SPLINE
SPL {X  -165.650, Y  +484.445, Z    +0.000, E1   +32.277, E3 +434870.647}
SPL {X  -165.650, Y  +481.524, Z    +0.000, E1   +31.089, E3 +434888.097}
SPL {X  -165.650, Y  +478.014, Z    +0.000, E1   +30.826, E3 +434901.705}
SPL {X  -165.650, Y  +474.473, Z    +0.000, E1   +30.943, E3 +434913.029}
SPL {X  -165.650, Y  +471.826, Z    +0.000, E1   +30.770, E3 +434923.213}
SPL {X  -165.650, Y  +467.753, Z    +0.000, E1   +30.878, E3 +434936.586}
SPL {X  -165.650, Y  +463.837, Z    +0.000, E1   +30.924, E3 +434949.520}
SPL {X  -165.650, Y  +461.106, Z    +0.000, E1   +30.916, E3 +434958.907}
SPL {X  -165.650, Y  +457.156, Z    +0.000, E1   +30.860, E3 +434972.984}
SPL {X  -165.650, Y  +453.156, Z    +0.000, E1   +30.934, E3 +434985.958}
SPL {X  -165.650, Y  +450.433, Z    +0.000, E1   +30.789, E3 +434996.313}
SPL {X  -165.650, Y  +447.097, Z    +0.000, E1   +30.843, E3 +435007.362}
SPL {X  -165.650, Y  +443.673, Z    +0.000, E1   +30.907, E3 +435018.669}
SPL {X  -165.650, Y  +439.486, Z    +0.000, E1   +30.857, E3 +435033.479}
SPL {X  -165.650, Y  +435.146, Z    +0.000, E1   +30.969, E3 +435047.398}
SPL {X  -165.650, Y  +431.607, Z    +0.000, E1   +30.889, E3 +435060.113}
SPL {X  -165.650, Y  +427.340, Z    +0.000, E1   +30.870, E3 +435074.824}
SPL {X  -165.650, Y  +423.901, Z    +0.000, E1   +30.858, E3 +435086.580}
SPL {X  -165.650, Y  +421.437, Z    +0.000, E1   +30.833, E3 +435095.179}
SPL {X  -165.650, Y  +418.489, Z    +0.000, E1   +30.835, E3 +435105.295}
SPL {X  -165.650, Y  +414.127, Z    +0.000, E1   +30.869, E3 +435120.204}
SPL {X  -165.650, Y  +408.547, Z    +0.000, E1   +30.964, E3 +435138.620}
SPL {X  -165.650, Y  +405.433, Z    +0.000, E1   +30.730, E3 +435150.597}
SPL {X  -165.650, Y  +401.473, Z    +0.000, E1   +30.933, E3 +435163.045}
SPL {X  -165.650, Y  +396.018, Z    +0.000, E1   +30.861, E3 +435182.230}
SPL {X  -165.650, Y  +390.331, Z    +0.000, E1   +30.892, E3 +435201.483}
SPL {X  -165.650, Y  +384.849, Z    +0.000, E1   +30.885, E3 +435220.286}
SPL {X  -165.650, Y  +380.752, Z    +0.000, E1   +30.927, E3 +435233.787}
SPL {X  -165.648, Y  +377.739, Z    +0.000, E1   +30.835, E3 +435244.797}
SPL {X  -165.594, Y  +374.183, Z    +0.000, E1   +30.878, E3 +435256.634}
SPL {X  -165.492, Y  +371.263, Z    +0.000, E1   +30.913, E3 +435266.329}
SPL {X  -165.379, Y  +369.027, Z    +0.000, E1   +30.727, E3 +435275.267}
SPL {X  -165.167, Y  +365.866, Z    +0.000, E1   +30.741, E3 +435286.041}
SPL {X  -164.892, Y  +362.671, Z    +0.000, E1   +30.830, E3 +435296.365}
SPL {X  -164.570, Y  +359.612, Z    +0.000, E1   +30.773, E3 +435307.178}
SPL {X  -164.104, Y  +355.923, Z    +0.000, E1   +30.626, E3 +435320.895}
SPL {X  -163.573, Y  +352.353, Z    +0.000, E1   +30.451, E3 +435334.159}
SPL {X  -162.476, Y  +346.230, Z    +0.000, E1   +31.677, E3 +435346.740}
SPL {X  -152.976, Y  +314.952, Z    +0.000, E1   +38.607, E3 +435395.705}
SPL {X  -137.967, Y  +286.821, Z    +0.000, E1   +43.969, E3 +435438.926}
ENDSPLINE

SPLINE
SPL {X  -153.316, Y  +315.777, Z    +0.000, E1   +33.140, E3 +435481.554}
SPL {X  -164.446, Y  +358.564, Z    +0.000, E1   +15.149, E3 +435446.765}
SPL {X  -165.379, Y  +369.025, Z    +0.000, E1    +9.158, E3 +435452.490}
SPL {X  -165.612, Y  +374.969, Z    +0.000, E1    +5.630, E3 +435455.165}
SPL {X  -165.650, Y  +383.362, Z    +0.000, E1    +0.177, E3 +435439.783}
SPL {X  -165.650, Y  +383.923, Z    +0.000, E1    -0.215, E3 +435452.941}
SPL {X  -165.650, Y  +388.083, Z    +0.000, E1    -3.355, E3 +435451.804}
SPL {X  -165.650, Y  +393.983, Z    +0.000, E1    -8.501, E3 +435448.203}
SPL {X  -165.650, Y  +402.241, Z    +0.000, E1   -16.711, E3 +435442.714}
SPL {X  -165.650, Y  +416.345, Z    +0.000, E1   -29.511, E3 +435442.506}
SPL {X  -165.650, Y  +422.331, Z    +0.000, E1   -27.760, E3 +435468.005}
SPL {X  -165.650, Y  +441.276, Z    +0.000, E1   -37.343, E3 +435477.862}
SPL {X  -165.650, Y  +462.890, Z    +0.000, E1   -40.484, E3 +435511.945}
ENDSPLINE

SPLINE
SPL {X  -165.650, Y  +446.920, Z    +0.000, E1   -31.238, E3 +435524.271}
ENDSPLINE

SPLINE
SPL {X  -165.650, Y  +447.935, Z    +0.000, E1   -30.213, E3 +435534.559}
SPL {X  -165.650, Y  +451.020, Z    +0.000, E1   -30.224, E3 +435545.379}
SPL {X  -165.650, Y  +454.519, Z    +0.000, E1   -30.374, E3 +435556.562}
SPL {X  -165.650, Y  +456.542, Z    +0.000, E1   -29.986, E3 +435566.306}
SPL {X  -165.650, Y  +460.618, Z    +0.000, E1   -30.298, E3 +435578.627}
SPL {X  -165.650, Y  +463.853, Z    +0.000, E1   -30.103, E3 +435591.228}
SPL {X  -165.650, Y  +467.246, Z    +0.000, E1   -30.279, E3 +435601.958}
SPL {X  -165.650, Y  +469.780, Z    +0.000, E1   -30.237, E3 +435611.083}
SPL {X  -165.650, Y  +472.566, Z    +0.000, E1   -30.124, E3 +435621.741}
SPL {X  -165.650, Y  +476.540, Z    +0.000, E1   -30.193, E3 +435635.285}
SPL {X  -165.650, Y  +480.320, Z    +0.000, E1   -30.163, E3 +435648.763}
SPL {X  -165.650, Y  +484.477, Z    +0.000, E1   -30.274, E3 +435662.652}
SPL {X  -165.650, Y  +488.041, Z    +0.000, E1   -30.253, E3 +435675.207}
SPL {X  -165.650, Y  +491.281, Z    +0.000, E1   -30.148, E3 +435687.345}
SPL {X  -165.650, Y  +495.051, Z    +0.000, E1   -30.213, E3 +435700.154}
SPL {X  -165.650, Y  +498.418, Z    +0.000, E1   -30.282, E3 +435711.447}
SPL {X  -165.650, Y  +500.833, Z    +0.000, E1   -30.191, E3 +435720.496}
SPL {X  -165.650, Y  +504.246, Z    +0.000, E1   -30.231, E3 +435732.362}
SPL {X  -165.650, Y  +507.017, Z    +0.000, E1   -30.108, E3 +435742.771}
SPL {X  -165.650, Y  +510.660, Z    +0.000, E1   -30.223, E3 +435755.037}
SPL {X  -165.650, Y  +515.918, Z    +0.000, E1   -30.316, E3 +435772.846}
SPL {X  -165.650, Y  +520.621, Z    +0.000, E1   -30.198, E3 +435790.131}
SPL {X  -165.650, Y  +525.344, Z    +0.000, E1   -30.269, E3 +435806.187}
SPL {X  -165.650, Y  +528.152, Z    +0.000, E1   -29.991, E3 +435817.828}
SPL {X  -165.650, Y  +531.783, Z    +0.000, E1   -30.416, E3 +435827.721}
SPL {X  -165.650, Y  +534.115, Z    +0.000, E1   -30.089, E3 +435838.103}
SPL {X  -165.650, Y  +538.363, Z    +0.000, E1   -30.232, E3 +435852.273}
SPL {X  -165.650, Y  +543.650, Z    +0.000, E1   -30.281, E3 +435870.493}
SPL {X  -165.650, Y  +547.199, Z    +0.000, E1   -30.132, E3 +435883.752}
SPL {X  -165.650, Y  +550.512, Z    +0.000, E1   -30.197, E3 +435895.078}
SPL {X  -165.650, Y  +554.908, Z    +0.000, E1   -30.180, E3 +435910.739}
SPL {X  -165.650, Y  +560.243, Z    +0.000, E1   -30.214, E3 +435929.365}
SPL {X  -165.650, Y  +565.528, Z    +0.000, E1   -30.192, E3 +435948.057}
SPL {X  -165.650, Y  +570.048, Z    +0.000, E1   -30.238, E3 +435963.488}
SPL {X  -165.650, Y  +573.110, Z    +0.000, E1   -30.057, E3 +435975.473}
SPL {X  -165.650, Y  +577.587, Z    +0.000, E1   -30.270, E3 +435989.912}
SPL {X  -165.650, Y  +581.190, Z    +0.000, E1   -30.107, E3 +436003.551}
SPL {X  -165.650, Y  +585.053, Z    +0.000, E1   -30.090, E3 +436017.422}
ENDSPLINE

SPLINE
SPL {X  -165.650, Y  +484.445, Z    +0.000, E1   +32.277, E3 +436034.826}
SPL {X  -165.650, Y  +481.524, Z    +0.000, E1   +31.089, E3 +436052.277}
SPL {X  -165.650, Y  +478.014, Z    +0.000, E1   +30.826, E3 +436065.884}
SPL {X  -165.650, Y  +474.473, Z    +0.000, E1   +30.943, E3 +436077.209}
SPL {X  -165.650, Y  +471.826, Z    +0.000, E1   +30.770, E3 +436087.392}
SPL {X  -165.650, Y  +467.753, Z    +0.000, E1   +30.878, E3 +436100.766}
SPL {X  -165.650, Y  +463.837, Z    +0.000, E1   +30.924, E3 +436113.699}
SPL {X  -165.650, Y  +461.106, Z    +0.000, E1   +30.916, E3 +436123.086}
SPL {X  -165.650, Y  +457.156, Z    +0.000, E1   +30.860, E3 +436137.163}
SPL {X  -165.650, Y  +453.156, Z    +0.000, E1   +30.934, E3 +436150.137}
SPL {X  -165.650, Y  +450.433, Z    +0.000, E1   +30.789, E3 +436160.492}
SPL {X  -165.650, Y  +447.097, Z    +0.000, E1   +30.843, E3 +436171.541}
SPL {X  -165.650, Y  +443.673, Z    +0.000, E1   +30.907, E3 +436182.848}
SPL {X  -165.650, Y  +439.486, Z    +0.000, E1   +30.857, E3 +436197.658}
SPL {X  -165.650, Y  +434.043, Z    +0.000, E1   +30.950, E3 +436215.674}
SPL {X  -165.650, Y  +430.419, Z    +0.000, E1   +30.895, E3 +436228.177}
SPL {X  -165.650, Y  +427.340, Z    +0.000, E1   +30.870, E3 +436239.003}
SPL {X  -165.650, Y  +422.641, Z    +0.000, E1   +30.884, E3 +436255.092}
SPL {X  -165.650, Y  +417.366, Z    +0.000, E1   +30.879, E3 +436273.198}
SPL {X  -165.650, Y  +412.139, Z    +0.000, E1   +30.870, E3 +436291.148}
SPL {X  -165.650, Y  +406.834, Z    +0.000, E1   +30.919, E3 +436308.976}
SPL {X  -165.650, Y  +402.516, Z    +0.000, E1   +30.874, E3 +436323.899}
SPL {X  -165.650, Y  +398.147, Z    +0.000, E1   +30.902, E3 +436338.777}
SPL {X  -165.650, Y  +394.694, Z    +0.000, E1   +30.805, E3 +436351.085}
SPL {X  -165.650, Y  +391.522, Z    +0.000, E1   +30.837, E3 +436361.766}
SPL {X  -165.650, Y  +387.533, Z    +0.000, E1   +30.858, E3 +436375.392}
SPL {X  -165.650, Y  +383.627, Z    +0.000, E1   +30.885, E3 +436388.453}
SPL {X  -165.650, Y  +380.752, Z    +0.000, E1   +30.927, E3 +436397.967}
SPL {X  -165.648, Y  +377.739, Z    +0.000, E1   +30.835, E3 +436408.976}
SPL {X  -165.594, Y  +374.183, Z    +0.000, E1   +30.878, E3 +436420.813}
SPL {X  -165.492, Y  +371.263, Z    +0.000, E1   +30.913, E3 +436430.508}
SPL {X  -165.379, Y  +369.027, Z    +0.000, E1   +30.727, E3 +436439.446}
SPL {X  -165.167, Y  +365.866, Z    +0.000, E1   +30.741, E3 +436450.220}
SPL {X  -164.892, Y  +362.671, Z    +0.000, E1   +30.830, E3 +436460.545}
SPL {X  -164.570, Y  +359.612, Z    +0.000, E1   +30.773, E3 +436471.357}
SPL {X  -164.104, Y  +355.923, Z    +0.000, E1   +30.626, E3 +436485.074}
SPL {X  -163.573, Y  +352.353, Z    +0.000, E1   +30.451, E3 +436498.338}
SPL {X  -162.476, Y  +346.230, Z    +0.000, E1   +31.677, E3 +436510.919}
SPL {X  -152.976, Y  +314.952, Z    +0.000, E1   +38.607, E3 +436559.884}
SPL {X  -137.967, Y  +286.821, Z    +0.000, E1   +43.969, E3 +436603.106}
ENDSPLINE

SPLINE
SPL {X  -153.316, Y  +315.777, Z    +0.000, E1   +33.140, E3 +436645.733}
SPL {X  -164.446, Y  +358.564, Z    +0.000, E1   +15.149, E3 +436610.944}
SPL {X  -165.379, Y  +369.025, Z    +0.000, E1    +9.158, E3 +436616.669}
SPL {X  -165.612, Y  +374.969, Z    +0.000, E1    +5.630, E3 +436619.344}
SPL {X  -165.650, Y  +383.362, Z    +0.000, E1    +0.177, E3 +436603.963}
SPL {X  -165.650, Y  +383.923, Z    +0.000, E1    -0.215, E3 +436617.120}
SPL {X  -165.650, Y  +388.083, Z    +0.000, E1    -3.355, E3 +436615.983}
SPL {X  -165.650, Y  +393.983, Z    +0.000, E1    -8.501, E3 +436612.382}
SPL {X  -165.650, Y  +402.241, Z    +0.000, E1   -16.711, E3 +436606.893}
SPL {X  -165.650, Y  +416.345, Z    +0.000, E1   -29.511, E3 +436606.685}
SPL {X  -165.650, Y  +422.331, Z    +0.000, E1   -27.760, E3 +436632.184}
SPL {X  -165.650, Y  +441.276, Z    +0.000, E1   -37.343, E3 +436642.042}
SPL {X  -165.650, Y  +462.890, Z    +0.000, E1   -40.484, E3 +436676.124}
ENDSPLINE

SPLINE
SPL {X  -165.650, Y  +446.920, Z    +0.000, E1   -31.238, E3 +436688.450}
ENDSPLINE

SPLINE
SPL {X  -165.650, Y  +447.935, Z    +0.000, E1   -30.213, E3 +436698.738}
SPL {X  -165.650, Y  +451.020, Z    +0.000, E1   -30.224, E3 +436709.559}
SPL {X  -165.650, Y  +454.519, Z    +0.000, E1   -30.374, E3 +436720.741}
SPL {X  -165.650, Y  +457.429, Z    +0.000, E1   -30.029, E3 +436733.443}
SPL {X  -165.650, Y  +461.678, Z    +0.000, E1   -30.426, E3 +436745.567}
SPL {X  -165.650, Y  +463.853, Z    +0.000, E1   -30.103, E3 +436755.407}
SPL {X  -165.650, Y  +468.397, Z    +0.000, E1   -30.302, E3 +436770.211}
SPL {X  -165.650, Y  +472.566, Z    +0.000, E1   -30.124, E3 +436785.920}
SPL {X  -165.650, Y  +476.540, Z    +0.000, E1   -30.193, E3 +436799.464}
SPL {X  -165.650, Y  +481.042, Z    +0.000, E1   -30.192, E3 +436815.409}
SPL {X  -165.650, Y  +485.236, Z    +0.000, E1   -30.294, E3 +436829.265}
SPL {X  -165.650, Y  +489.057, Z    +0.000, E1   -30.341, E3 +436842.471}
SPL {X  -165.650, Y  +491.647, Z    +0.000, E1   -29.894, E3 +436854.404}
SPL {X  -165.650, Y  +495.051, Z    +0.000, E1   -30.213, E3 +436864.333}
SPL {X  -165.650, Y  +498.418, Z    +0.000, E1   -30.282, E3 +436875.626}
SPL {X  -165.650, Y  +502.421, Z    +0.000, E1   -30.263, E3 +436889.983}
SPL {X  -165.650, Y  +506.344, Z    +0.000, E1   -30.129, E3 +436904.513}
SPL {X  -165.650, Y  +509.866, Z    +0.000, E1   -30.236, E3 +436916.182}
SPL {X  -165.650, Y  +513.685, Z    +0.000, E1   -30.234, E3 +436929.679}
SPL {X  -165.650, Y  +517.919, Z    +0.000, E1   -30.227, E3 +436944.586}
SPL {X  -165.650, Y  +521.521, Z    +0.000, E1   -30.210, E3 +436957.260}
SPL {X  -165.650, Y  +525.344, Z    +0.000, E1   -30.269, E3 +436970.367}
SPL {X  -165.650, Y  +528.152, Z    +0.000, E1   -29.991, E3 +436982.008}
SPL {X  -165.650, Y  +531.783, Z    +0.000, E1   -30.416, E3 +436991.900}
SPL {X  -165.650, Y  +534.115, Z    +0.000, E1   -30.089, E3 +437002.282}
SPL {X  -165.650, Y  +538.363, Z    +0.000, E1   -30.232, E3 +437016.452}
SPL {X  -165.650, Y  +543.650, Z    +0.000, E1   -30.281, E3 +437034.672}
SPL {X  -165.650, Y  +547.199, Z    +0.000, E1   -30.132, E3 +437047.931}
SPL {X  -165.650, Y  +550.512, Z    +0.000, E1   -30.197, E3 +437059.257}
SPL {X  -165.650, Y  +554.908, Z    +0.000, E1   -30.180, E3 +437074.918}
SPL {X  -165.650, Y  +560.243, Z    +0.000, E1   -30.214, E3 +437093.544}
SPL {X  -165.650, Y  +565.528, Z    +0.000, E1   -30.192, E3 +437112.236}
SPL {X  -165.650, Y  +570.048, Z    +0.000, E1   -30.238, E3 +437127.667}
SPL {X  -165.650, Y  +573.110, Z    +0.000, E1   -30.057, E3 +437139.652}
SPL {X  -165.650, Y  +577.587, Z    +0.000, E1   -30.270, E3 +437154.091}
SPL {X  -165.650, Y  +581.190, Z    +0.000, E1   -30.107, E3 +437167.731}
SPL {X  -165.650, Y  +585.053, Z    +0.000, E1   -30.090, E3 +437181.601}
ENDSPLINE

SPLINE
SPL {X  -165.650, Y  +484.445, Z    +0.000, E1   +32.277, E3 +437199.005}
SPL {X  -165.650, Y  +481.524, Z    +0.000, E1   +31.089, E3 +437216.456}
SPL {X  -165.650, Y  +478.014, Z    +0.000, E1   +30.826, E3 +437230.063}
SPL {X  -165.650, Y  +474.473, Z    +0.000, E1   +30.943, E3 +437241.388}
SPL {X  -165.650, Y  +471.826, Z    +0.000, E1   +30.770, E3 +437251.571}
SPL {X  -165.650, Y  +467.753, Z    +0.000, E1   +30.878, E3 +437264.945}
SPL {X  -165.650, Y  +463.837, Z    +0.000, E1   +30.924, E3 +437277.878}
SPL {X  -165.650, Y  +461.106, Z    +0.000, E1   +30.916, E3 +437287.265}
SPL {X  -165.650, Y  +457.156, Z    +0.000, E1   +30.860, E3 +437301.342}
SPL {X  -165.650, Y  +453.156, Z    +0.000, E1   +30.934, E3 +437314.316}
SPL {X  -165.650, Y  +450.433, Z    +0.000, E1   +30.789, E3 +437324.671}
SPL {X  -165.650, Y  +447.097, Z    +0.000, E1   +30.843, E3 +437335.720}
SPL {X  -165.650, Y  +443.673, Z    +0.000, E1   +30.907, E3 +437347.027}
SPL {X  -165.650, Y  +439.486, Z    +0.000, E1   +30.857, E3 +437361.837}
SPL {X  -165.650, Y  +435.146, Z    +0.000, E1   +30.969, E3 +437375.756}
SPL {X  -165.650, Y  +432.765, Z    +0.000, E1   +30.831, E3 +437384.771}
SPL {X  -165.650, Y  +429.309, Z    +0.000, E1   +30.920, E3 +437396.111}
SPL {X  -165.650, Y  +424.918, Z    +0.000, E1   +30.862, E3 +437411.569}
SPL {X  -165.650, Y  +421.437, Z    +0.000, E1   +30.833, E3 +437423.537}
SPL {X  -165.650, Y  +418.489, Z    +0.000, E1   +30.835, E3 +437433.654}
SPL {X  -165.650, Y  +415.831, Z    +0.000, E1   +30.847, E3 +437442.616}
SPL {X  -165.650, Y  +412.139, Z    +0.000, E1   +30.870, E3 +437455.327}
SPL {X  -165.650, Y  +406.834, Z    +0.000, E1   +30.919, E3 +437473.156}
SPL {X  -165.650, Y  +402.516, Z    +0.000, E1   +30.874, E3 +437488.078}
SPL {X  -165.650, Y  +398.147, Z    +0.000, E1   +30.902, E3 +437502.956}
SPL {X  -165.650, Y  +394.694, Z    +0.000, E1   +30.805, E3 +437515.265}
SPL {X  -165.650, Y  +391.522, Z    +0.000, E1   +30.837, E3 +437525.945}
SPL {X  -165.650, Y  +387.533, Z    +0.000, E1   +30.858, E3 +437539.572}
SPL {X  -165.650, Y  +383.627, Z    +0.000, E1   +30.885, E3 +437552.632}
SPL {X  -165.650, Y  +380.752, Z    +0.000, E1   +30.927, E3 +437562.146}
SPL {X  -165.648, Y  +377.739, Z    +0.000, E1   +30.835, E3 +437573.155}
SPL {X  -165.594, Y  +374.183, Z    +0.000, E1   +30.878, E3 +437584.992}
SPL {X  -165.429, Y  +369.945, Z    +0.000, E1   +30.850, E3 +437599.867}
SPL {X  -165.167, Y  +365.866, Z    +0.000, E1   +30.741, E3 +437614.400}
SPL {X  -164.892, Y  +362.671, Z    +0.000, E1   +30.830, E3 +437624.724}
SPL {X  -164.570, Y  +359.612, Z    +0.000, E1   +30.773, E3 +437635.536}
SPL {X  -164.104, Y  +355.923, Z    +0.000, E1   +30.626, E3 +437649.253}
SPL {X  -163.573, Y  +352.353, Z    +0.000, E1   +30.451, E3 +437662.518}
SPL {X  -162.476, Y  +346.230, Z    +0.000, E1   +31.677, E3 +437675.098}
SPL {X  -152.976, Y  +314.952, Z    +0.000, E1   +38.607, E3 +437724.064}
SPL {X  -137.967, Y  +286.821, Z    +0.000, E1   +43.969, E3 +437767.285}
ENDSPLINE

SPLINE
SPL {X  -153.316, Y  +315.777, Z    +0.000, E1   +33.140, E3 +437809.912}
SPL {X  -164.446, Y  +358.564, Z    +0.000, E1   +15.149, E3 +437775.123}
SPL {X  -165.510, Y  +371.680, Z    +0.000, E1    +7.684, E3 +437779.179}
SPL {X  -165.628, Y  +375.818, Z    +0.000, E1    +5.016, E3 +437787.108}
SPL {X  -165.650, Y  +383.362, Z    +0.000, E1    +0.177, E3 +437768.142}
SPL {X  -165.650, Y  +383.923, Z    +0.000, E1    -0.215, E3 +437781.299}
SPL {X  -165.650, Y  +388.083, Z    +0.000, E1    -3.355, E3 +437780.163}
SPL {X  -165.650, Y  +395.510, Z    +0.000, E1    -9.810, E3 +437776.289}
SPL {X  -165.650, Y  +403.066, Z    +0.000, E1   -17.886, E3 +437769.122}
SPL {X  -165.650, Y  +416.345, Z    +0.000, E1   -29.511, E3 +437770.864}
SPL {X  -165.650, Y  +422.331, Z    +0.000, E1   -27.760, E3 +437796.364}
SPL {X  -165.650, Y  +435.050, Z    +0.000, E1   -34.610, E3 +437802.866}
SPL {X  -165.650, Y  +446.725, Z    +0.000, E1   -39.593, E3 +437809.127}
SPL {X  -165.650, Y  +462.890, Z    +0.000, E1   -40.484, E3 +437840.304}
ENDSPLINE

SPLINE
SPL {X  -165.650, Y  +446.920, Z    +0.000, E1   -31.238, E3 +437852.629}
ENDSPLINE

SPLINE
SPL {X  -165.650, Y  +447.935, Z    +0.000, E1   -30.213, E3 +437862.917}
SPL {X  -165.650, Y  +451.020, Z    +0.000, E1   -30.224, E3 +437873.738}
SPL {X  -165.650, Y  +454.519, Z    +0.000, E1   -30.374, E3 +437884.920}
SPL {X  -165.650, Y  +457.429, Z    +0.000, E1   -30.029, E3 +437897.622}
SPL {X  -165.650, Y  +461.678, Z    +0.000, E1   -30.426, E3 +437909.746}
SPL {X  -165.650, Y  +463.853, Z    +0.000, E1   -30.103, E3 +437919.586}
SPL {X  -165.650, Y  +468.397, Z    +0.000, E1   -30.302, E3 +437934.390}
SPL {X  -165.650, Y  +472.566, Z    +0.000, E1   -30.124, E3 +437950.099}
SPL {X  -165.650, Y  +476.540, Z    +0.000, E1   -30.193, E3 +437963.643}
SPL {X  -165.650, Y  +481.042, Z    +0.000, E1   -30.192, E3 +437979.589}
SPL {X  -165.650, Y  +485.236, Z    +0.000, E1   -30.294, E3 +437993.444}
SPL {X  -165.650, Y  +489.057, Z    +0.000, E1   -30.341, E3 +438006.650}
SPL {X  -165.650, Y  +491.647, Z    +0.000, E1   -29.894, E3 +438018.583}
SPL {X  -165.650, Y  +495.051, Z    +0.000, E1   -30.213, E3 +438028.512}
SPL {X  -165.650, Y  +498.418, Z    +0.000, E1   -30.282, E3 +438039.805}
SPL {X  -165.650, Y  +502.421, Z    +0.000, E1   -30.263, E3 +438054.162}
SPL {X  -165.650, Y  +506.344, Z    +0.000, E1   -30.129, E3 +438068.692}
SPL {X  -165.650, Y  +509.866, Z    +0.000, E1   -30.236, E3 +438080.361}
SPL {X  -165.650, Y  +513.685, Z    +0.000, E1   -30.234, E3 +438093.858}
SPL {X  -165.650, Y  +517.919, Z    +0.000, E1   -30.227, E3 +438108.765}
SPL {X  -165.650, Y  +521.521, Z    +0.000, E1   -30.210, E3 +438121.439}
SPL {X  -165.650, Y  +525.344, Z    +0.000, E1   -30.269, E3 +438134.546}
SPL {X  -165.650, Y  +528.152, Z    +0.000, E1   -29.991, E3 +438146.187}
SPL {X  -165.650, Y  +531.783, Z    +0.000, E1   -30.416, E3 +438156.079}
SPL {X  -165.650, Y  +534.115, Z    +0.000, E1   -30.089, E3 +438166.462}
SPL {X  -165.650, Y  +537.522, Z    +0.000, E1   -30.251, E3 +438177.376}
SPL {X  -165.650, Y  +540.621, Z    +0.000, E1   -30.014, E3 +438189.937}
SPL {X  -165.650, Y  +544.944, Z    +0.000, E1   -30.447, E3 +438202.136}
SPL {X  -165.650, Y  +548.549, Z    +0.000, E1   -30.216, E3 +438216.460}
SPL {X  -165.650, Y  +553.092, Z    +0.000, E1   -30.157, E3 +438232.802}
SPL {X  -165.650, Y  +557.277, Z    +0.000, E1   -30.150, E3 +438247.551}
SPL {X  -165.650, Y  +561.168, Z    +0.000, E1   -30.194, E3 +438260.932}
SPL {X  -165.650, Y  +564.449, Z    +0.000, E1   -30.167, E3 +438272.616}
SPL {X  -165.650, Y  +566.935, Z    +0.000, E1   -30.135, E3 +438281.521}
SPL {X  -165.650, Y  +570.048, Z    +0.000, E1   -30.238, E3 +438291.846}
SPL {X  -165.650, Y  +573.110, Z    +0.000, E1   -30.057, E3 +438303.831}
SPL {X  -165.650, Y  +577.587, Z    +0.000, E1   -30.270, E3 +438318.270}
SPL {X  -165.650, Y  +581.190, Z    +0.000, E1   -30.107, E3 +438331.910}
SPL {X  -165.650, Y  +585.053, Z    +0.000, E1   -30.090, E3 +438345.780}
ENDSPLINE

SPLINE
SPL {X  -165.650, Y  +484.445, Z    +0.000, E1   +32.277, E3 +438363.184}
SPL {X  -165.650, Y  +481.524, Z    +0.000, E1   +31.089, E3 +438380.635}
SPL {X  -165.650, Y  +478.014, Z    +0.000, E1   +30.826, E3 +438394.242}
SPL {X  -165.650, Y  +474.473, Z    +0.000, E1   +30.943, E3 +438405.567}
SPL {X  -165.650, Y  +471.826, Z    +0.000, E1   +30.770, E3 +438415.750}
SPL {X  -165.650, Y  +467.753, Z    +0.000, E1   +30.878, E3 +438429.124}
SPL {X  -165.650, Y  +463.837, Z    +0.000, E1   +30.924, E3 +438442.058}
SPL {X  -165.650, Y  +461.106, Z    +0.000, E1   +30.916, E3 +438451.445}
SPL {X  -165.650, Y  +458.435, Z    +0.000, E1   +30.759, E3 +438461.653}
SPL {X  -165.650, Y  +454.220, Z    +0.000, E1   +30.954, E3 +438474.886}
SPL {X  -165.650, Y  +450.433, Z    +0.000, E1   +30.789, E3 +438488.850}
SPL {X  -165.650, Y  +447.097, Z    +0.000, E1   +30.843, E3 +438499.899}
SPL {X  -165.650, Y  +443.673, Z    +0.000, E1   +30.907, E3 +438511.207}
SPL {X  -165.650, Y  +440.976, Z    +0.000, E1   +30.719, E3 +438521.663}
SPL {X  -165.650, Y  +437.973, Z    +0.000, E1   +30.928, E3 +438530.536}
SPL {X  -165.650, Y  +434.043, Z    +0.000, E1   +30.950, E3 +438544.032}
SPL {X  -165.650, Y  +430.419, Z    +0.000, E1   +30.895, E3 +438556.535}
SPL {X  -165.650, Y  +427.340, Z    +0.000, E1   +30.870, E3 +438567.362}
SPL {X  -165.650, Y  +422.641, Z    +0.000, E1   +30.884, E3 +438583.451}
SPL {X  -165.650, Y  +418.489, Z    +0.000, E1   +30.835, E3 +438597.833}
SPL {X  -165.650, Y  +414.127, Z    +0.000, E1   +30.869, E3 +438612.741}
SPL {X  -165.650, Y  +408.547, Z    +0.000, E1   +30.964, E3 +438631.157}
SPL {X  -165.650, Y  +405.433, Z    +0.000, E1   +30.730, E3 +438643.134}
SPL {X  -165.650, Y  +401.473, Z    +0.000, E1   +30.933, E3 +438655.583}
SPL {X  -165.650, Y  +396.018, Z    +0.000, E1   +30.861, E3 +438674.767}
SPL {X  -165.650, Y  +391.522, Z    +0.000, E1   +30.837, E3 +438690.124}
SPL {X  -165.650, Y  +387.533, Z    +0.000, E1   +30.858, E3 +438703.751}
SPL {X  -165.650, Y  +383.627, Z    +0.000, E1   +30.885, E3 +438716.811}
SPL {X  -165.650, Y  +380.752, Z    +0.000, E1   +30.927, E3 +438726.325}
SPL {X  -165.648, Y  +377.739, Z    +0.000, E1   +30.835, E3 +438737.334}
SPL {X  -165.594, Y  +374.183, Z    +0.000, E1   +30.878, E3 +438749.171}
SPL {X  -165.429, Y  +369.945, Z    +0.000, E1   +30.850, E3 +438764.046}
SPL {X  -165.167, Y  +365.866, Z    +0.000, E1   +30.741, E3 +438778.579}
SPL {X  -164.892, Y  +362.671, Z    +0.000, E1   +30.830, E3 +438788.903}
SPL {X  -164.570, Y  +359.612, Z    +0.000, E1   +30.773, E3 +438799.715}
SPL {X  -164.287, Y  +357.291, Z    +0.000, E1   +30.513, E3 +438809.345}
SPL {X  -163.720, Y  +353.284, Z    +0.000, E1   +30.592, E3 +438822.792}
SPL {X  -162.976, Y  +348.856, Z    +0.000, E1   +30.757, E3 +438836.620}
SPL {X  -161.497, Y  +341.640, Z    +0.000, E1   +33.276, E3 +438843.898}
SPL {X  -152.976, Y  +314.952, Z    +0.000, E1   +38.607, E3 +438888.243}
SPL {X  -137.967, Y  +286.821, Z    +0.000, E1   +43.969, E3 +438931.464}
ENDSPLINE

SPLINE
SPL {X  -149.143, Y  +306.414, Z    +0.000, E1   +36.361, E3 +438982.596}
SPL {X  -163.091, Y  +349.496, Z    +0.000, E1   +19.699, E3 +438939.379}
SPL {X  -165.027, Y  +364.142, Z    +0.000, E1   +12.054, E3 +438942.520}
SPL {X  -165.612, Y  +374.969, Z    +0.000, E1    +5.630, E3 +438947.702}
SPL {X  -165.650, Y  +383.362, Z    +0.000, E1    +0.177, E3 +438932.321}
SPL {X  -165.650, Y  +383.923, Z    +0.000, E1    -0.215, E3 +438945.478}
SPL {X  -165.650, Y  +388.083, Z    +0.000, E1    -3.355, E3 +438944.342}
SPL {X  -165.650, Y  +395.510, Z    +0.000, E1    -9.810, E3 +438940.468}
SPL {X  -165.650, Y  +403.066, Z    +0.000, E1   -17.886, E3 +438933.301}
SPL {X  -165.650, Y  +414.811, Z    +0.000, E1   -28.314, E3 +438934.782}
SPL {X  -165.650, Y  +423.479, Z    +0.000, E1   -29.012, E3 +438958.711}
SPL {X  -165.650, Y  +441.276, Z    +0.000, E1   -37.343, E3 +438970.400}
SPL {X  -165.650, Y  +462.890, Z    +0.000, E1   -40.484, E3 +439004.483}
ENDSPLINE

SPLINE
SPL {X  -165.650, Y  +446.920, Z    +0.000, E1   -31.238, E3 +439016.808}
ENDSPLINE

SPLINE
SPL {X  -165.650, Y  +447.935, Z    +0.000, E1   -30.213, E3 +439027.096}
SPL {X  -165.650, Y  +451.020, Z    +0.000, E1   -30.224, E3 +439037.917}
SPL {X  -165.650, Y  +454.519, Z    +0.000, E1   -30.374, E3 +439049.099}
SPL {X  -165.650, Y  +456.542, Z    +0.000, E1   -29.986, E3 +439058.844}
SPL {X  -165.650, Y  +460.618, Z    +0.000, E1   -30.298, E3 +439071.164}
SPL {X  -165.650, Y  +463.853, Z    +0.000, E1   -30.103, E3 +439083.765}
SPL {X  -165.650, Y  +468.397, Z    +0.000, E1   -30.302, E3 +439098.569}
SPL {X  -165.650, Y  +472.566, Z    +0.000, E1   -30.124, E3 +439114.278}
SPL {X  -165.650, Y  +475.265, Z    +0.000, E1   -30.034, E3 +439124.316}
SPL {X  -165.650, Y  +479.559, Z    +0.000, E1   -30.258, E3 +439138.180}
SPL {X  -165.650, Y  +484.477, Z    +0.000, E1   -30.274, E3 +439155.189}
SPL {X  -165.650, Y  +488.041, Z    +0.000, E1   -30.253, E3 +439167.745}
SPL {X  -165.650, Y  +491.281, Z    +0.000, E1   -30.148, E3 +439179.883}
SPL {X  -165.650, Y  +495.051, Z    +0.000, E1   -30.213, E3 +439192.691}
SPL {X  -165.650, Y  +499.546, Z    +0.000, E1   -30.283, E3 +439208.134}
SPL {X  -165.650, Y  +503.544, Z    +0.000, E1   -30.247, E3 +439222.203}
SPL {X  -165.650, Y  +506.344, Z    +0.000, E1   -30.129, E3 +439232.871}
SPL {X  -165.650, Y  +509.866, Z    +0.000, E1   -30.236, E3 +439244.540}
SPL {X  -165.650, Y  +513.685, Z    +0.000, E1   -30.234, E3 +439258.037}
SPL {X  -165.650, Y  +517.919, Z    +0.000, E1   -30.227, E3 +439272.944}
SPL {X  -165.650, Y  +521.521, Z    +0.000, E1   -30.210, E3 +439285.619}
SPL {X  -165.650, Y  +525.344, Z    +0.000, E1   -30.269, E3 +439298.725}
SPL {X  -165.650, Y  +528.152, Z    +0.000, E1   -29.991, E3 +439310.366}
SPL {X  -165.650, Y  +531.783, Z    +0.000, E1   -30.416, E3 +439320.259}
SPL {X  -165.650, Y  +534.115, Z    +0.000, E1   -30.089, E3 +439330.641}
SPL {X  -165.650, Y  +537.522, Z    +0.000, E1   -30.251, E3 +439341.555}
SPL {X  -165.650, Y  +540.621, Z    +0.000, E1   -30.014, E3 +439354.116}
SPL {X  -165.650, Y  +544.944, Z    +0.000, E1   -30.447, E3 +439366.316}
SPL {X  -165.650, Y  +547.199, Z    +0.000, E1   -30.132, E3 +439376.289}
SPL {X  -165.650, Y  +550.512, Z    +0.000, E1   -30.197, E3 +439387.615}
SPL {X  -165.650, Y  +553.852, Z    +0.000, E1   -30.156, E3 +439399.556}
SPL {X  -165.650, Y  +557.277, Z    +0.000, E1   -30.150, E3 +439411.730}
SPL {X  -165.650, Y  +561.168, Z    +0.000, E1   -30.194, E3 +439425.112}
SPL {X  -165.650, Y  +565.528, Z    +0.000, E1   -30.192, E3 +439440.594}
SPL {X  -165.650, Y  +570.048, Z    +0.000, E1   -30.238, E3 +439456.025}
SPL {X  -165.650, Y  +573.110, Z    +0.000, E1   -30.057, E3 +439468.010}
SPL {X  -165.650, Y  +577.587, Z    +0.000, E1   -30.270, E3 +439482.449}
SPL {X  -165.650, Y  +581.190, Z    +0.000, E1   -30.107, E3 +439496.089}
SPL {X  -165.650, Y  +585.053, Z    +0.000, E1   -30.090, E3 +439509.959}
ENDSPLINE

SPLINE
SPL {X  -165.650, Y  +484.445, Z    +0.000, E1   +32.277, E3 +439527.363}
SPL {X  -165.650, Y  +481.524, Z    +0.000, E1   +31.089, E3 +439544.814}
SPL {X  -165.650, Y  +478.014, Z    +0.000, E1   +30.826, E3 +439558.421}
SPL {X  -165.650, Y  +474.473, Z    +0.000, E1   +30.943, E3 +439569.746}
SPL {X  -165.650, Y  +471.826, Z    +0.000, E1   +30.770, E3 +439579.929}
SPL {X  -165.650, Y  +467.753, Z    +0.000, E1   +30.878, E3 +439593.303}
SPL {X  -165.650, Y  +463.837, Z    +0.000, E1   +30.924, E3 +439606.237}
SPL {X  -165.650, Y  +461.106, Z    +0.000, E1   +30.916, E3 +439615.624}
SPL {X  -165.650, Y  +457.156, Z    +0.000, E1   +30.860, E3 +439629.700}
SPL {X  -165.650, Y  +453.156, Z    +0.000, E1   +30.934, E3 +439642.674}
SPL {X  -165.650, Y  +450.433, Z    +0.000, E1   +30.789, E3 +439653.030}
SPL {X  -165.650, Y  +447.097, Z    +0.000, E1   +30.843, E3 +439664.078}
SPL {X  -165.650, Y  +443.673, Z    +0.000, E1   +30.907, E3 +439675.386}
SPL {X  -165.650, Y  +439.486, Z    +0.000, E1   +30.857, E3 +439690.195}
SPL {X  -165.650, Y  +435.146, Z    +0.000, E1   +30.969, E3 +439704.114}
SPL {X  -165.650, Y  +432.765, Z    +0.000, E1   +30.831, E3 +439713.129}
SPL {X  -165.650, Y  +429.309, Z    +0.000, E1   +30.920, E3 +439724.470}
SPL {X  -165.650, Y  +424.918, Z    +0.000, E1   +30.862, E3 +439739.927}
SPL {X  -165.650, Y  +421.437, Z    +0.000, E1   +30.833, E3 +439751.895}
SPL {X  -165.650, Y  +417.366, Z    +0.000, E1   +30.879, E3 +439765.736}
SPL {X  -165.650, Y  +413.181, Z    +0.000, E1   +30.815, E3 +439780.333}
SPL {X  -165.650, Y  +408.547, Z    +0.000, E1   +30.964, E3 +439795.336}
SPL {X  -165.650, Y  +405.433, Z    +0.000, E1   +30.730, E3 +439807.313}
SPL {X  -165.650, Y  +402.516, Z    +0.000, E1   +30.874, E3 +439816.436}
SPL {X  -165.650, Y  +398.147, Z    +0.000, E1   +30.902, E3 +439831.314}
SPL {X  -165.650, Y  +394.694, Z    +0.000, E1   +30.805, E3 +439843.623}
SPL {X  -165.650, Y  +391.522, Z    +0.000, E1   +30.837, E3 +439854.304}
SPL {X  -165.650, Y  +387.533, Z    +0.000, E1   +30.858, E3 +439867.930}
SPL {X  -165.650, Y  +383.627, Z    +0.000, E1   +30.885, E3 +439880.990}
SPL {X  -165.650, Y  +380.752, Z    +0.000, E1   +30.927, E3 +439890.504}
SPL {X  -165.648, Y  +377.739, Z    +0.000, E1   +30.835, E3 +439901.513}
SPL {X  -165.594, Y  +374.183, Z    +0.000, E1   +30.878, E3 +439913.350}
SPL {X  -165.429, Y  +369.945, Z    +0.000, E1   +30.850, E3 +439928.225}
SPL {X  -165.167, Y  +365.866, Z    +0.000, E1   +30.741, E3 +439942.758}
SPL {X  -164.892, Y  +362.671, Z    +0.000, E1   +30.830, E3 +439953.082}
SPL {X  -164.570, Y  +359.612, Z    +0.000, E1   +30.773, E3 +439963.895}
SPL {X  -164.104, Y  +355.923, Z    +0.000, E1   +30.626, E3 +439977.611}
SPL {X  -163.573, Y  +352.353, Z    +0.000, E1   +30.451, E3 +439990.876}
SPL {X  -162.476, Y  +346.230, Z    +0.000, E1   +31.677, E3 +440003.457}
SPL {X  -152.976, Y  +314.952, Z    +0.000, E1   +38.607, E3 +440052.422}
SPL {X  -137.967, Y  +286.821, Z    +0.000, E1   +43.969, E3 +440095.643}
ENDSPLINE

SPLINE
SPL {X  -149.143, Y  +306.414, Z    +0.000, E1   +36.361, E3 +440146.775}
SPL {X  -164.268, Y  +357.145, Z    +0.000, E1   +15.880, E3 +440104.534}
SPL {X  -165.379, Y  +369.025, Z    +0.000, E1    +9.158, E3 +440109.206}
SPL {X  -165.612, Y  +374.969, Z    +0.000, E1    +5.630, E3 +440111.881}
SPL {X  -165.650, Y  +383.362, Z    +0.000, E1    +0.177, E3 +440096.500}
SPL {X  -165.650, Y  +383.923, Z    +0.000, E1    -0.215, E3 +440109.657}
SPL {X  -165.650, Y  +388.083, Z    +0.000, E1    -3.355, E3 +440108.521}
SPL {X  -165.650, Y  +393.983, Z    +0.000, E1    -8.501, E3 +440104.919}
SPL {X  -165.650, Y  +402.241, Z    +0.000, E1   -16.711, E3 +440099.431}
SPL {X  -165.650, Y  +416.345, Z    +0.000, E1   -29.511, E3 +440099.223}
SPL {X  -165.650, Y  +422.331, Z    +0.000, E1   -27.760, E3 +440124.722}
SPL {X  -165.650, Y  +441.276, Z    +0.000, E1   -37.343, E3 +440134.579}
SPL {X  -165.650, Y  +462.890, Z    +0.000, E1   -40.484, E3 +440168.662}
ENDSPLINE

SPLINE
SPL {X  -165.650, Y  +446.920, Z    +0.000, E1   -31.238, E3 +440180.988}
ENDSPLINE

SPLINE
SPL {X  -165.650, Y  +447.935, Z    +0.000, E1   -30.213, E3 +440191.275}
SPL {X  -165.650, Y  +451.020, Z    +0.000, E1   -30.224, E3 +440202.096}
SPL {X  -165.650, Y  +454.519, Z    +0.000, E1   -30.374, E3 +440213.278}
SPL {X  -165.650, Y  +457.429, Z    +0.000, E1   -30.029, E3 +440225.980}
SPL {X  -165.650, Y  +461.678, Z    +0.000, E1   -30.426, E3 +440238.105}
SPL {X  -165.650, Y  +463.853, Z    +0.000, E1   -30.103, E3 +440247.944}
SPL {X  -165.650, Y  +468.397, Z    +0.000, E1   -30.302, E3 +440262.748}
SPL {X  -165.650, Y  +472.566, Z    +0.000, E1   -30.124, E3 +440278.457}
SPL {X  -165.650, Y  +475.265, Z    +0.000, E1   -30.034, E3 +440288.495}
SPL {X  -165.650, Y  +477.862, Z    +0.000, E1   -30.319, E3 +440295.686}
SPL {X  -165.650, Y  +481.042, Z    +0.000, E1   -30.192, E3 +440307.947}
SPL {X  -165.650, Y  +485.236, Z    +0.000, E1   -30.294, E3 +440321.802}
SPL {X  -165.650, Y  +488.041, Z    +0.000, E1   -30.253, E3 +440331.924}
SPL {X  -165.650, Y  +491.281, Z    +0.000, E1   -30.148, E3 +440344.062}
SPL {X  -165.650, Y  +495.051, Z    +0.000, E1   -30.213, E3 +440356.870}
SPL {X  -165.650, Y  +499.546, Z    +0.000, E1   -30.283, E3 +440372.313}
SPL {X  -165.650, Y  +503.544, Z    +0.000, E1   -30.247, E3 +440386.382}
SPL {X  -165.650, Y  +506.344, Z    +0.000, E1   -30.129, E3 +440397.050}
SPL {X  -165.650, Y  +509.866, Z    +0.000, E1   -30.236, E3 +440408.720}
SPL {X  -165.650, Y  +513.685, Z    +0.000, E1   -30.234, E3 +440422.216}
SPL {X  -165.650, Y  +517.919, Z    +0.000, E1   -30.227, E3 +440437.123}
SPL {X  -165.650, Y  +521.521, Z    +0.000, E1   -30.210, E3 +440449.798}
SPL {X  -165.650, Y  +525.344, Z    +0.000, E1   -30.269, E3 +440462.904}
SPL {X  -165.650, Y  +528.152, Z    +0.000, E1   -29.991, E3 +440474.545}
SPL {X  -165.650, Y  +531.783, Z    +0.000, E1   -30.416, E3 +440484.438}
SPL {X  -165.650, Y  +534.115, Z    +0.000, E1   -30.089, E3 +440494.820}
SPL {X  -165.650, Y  +537.522, Z    +0.000, E1   -30.251, E3 +440505.734}
SPL {X  -165.650, Y  +540.621, Z    +0.000, E1   -30.014, E3 +440518.295}
SPL {X  -165.650, Y  +544.944, Z    +0.000, E1   -30.447, E3 +440530.495}
SPL {X  -165.650, Y  +547.199, Z    +0.000, E1   -30.132, E3 +440540.468}
SPL {X  -165.650, Y  +550.512, Z    +0.000, E1   -30.197, E3 +440551.794}
SPL {X  -165.650, Y  +553.852, Z    +0.000, E1   -30.156, E3 +440563.735}
SPL {X  -165.650, Y  +557.277, Z    +0.000, E1   -30.150, E3 +440575.909}
SPL {X  -165.650, Y  +561.168, Z    +0.000, E1   -30.194, E3 +440589.291}
SPL {X  -165.650, Y  +564.449, Z    +0.000, E1   -30.167, E3 +440600.974}
SPL {X  -165.650, Y  +566.935, Z    +0.000, E1   -30.135, E3 +440609.879}
SPL {X  -165.650, Y  +570.048, Z    +0.000, E1   -30.238, E3 +440620.205}
SPL {X  -165.650, Y  +573.110, Z    +0.000, E1   -30.057, E3 +440632.189}
SPL {X  -165.650, Y  +577.587, Z    +0.000, E1   -30.270, E3 +440646.628}
SPL {X  -165.650, Y  +581.190, Z    +0.000, E1   -30.107, E3 +440660.268}
SPL {X  -165.650, Y  +585.053, Z    +0.000, E1   -30.090, E3 +440674.138}
ENDSPLINE

SPLINE
SPL {X  -165.650, Y  +484.445, Z    +0.000, E1   +32.277, E3 +440691.542}
SPL {X  -165.650, Y  +481.524, Z    +0.000, E1   +31.089, E3 +440708.993}
SPL {X  -165.650, Y  +478.014, Z    +0.000, E1   +30.826, E3 +440722.601}
SPL {X  -165.650, Y  +474.473, Z    +0.000, E1   +30.943, E3 +440733.925}
SPL {X  -165.650, Y  +471.826, Z    +0.000, E1   +30.770, E3 +440744.109}
SPL {X  -165.650, Y  +467.753, Z    +0.000, E1   +30.878, E3 +440757.482}
SPL {X  -165.650, Y  +463.837, Z    +0.000, E1   +30.924, E3 +440770.416}
SPL {X  -165.650, Y  +461.106, Z    +0.000, E1   +30.916, E3 +440779.803}
SPL {X  -165.650, Y  +457.156, Z    +0.000, E1   +30.860, E3 +440793.879}
SPL {X  -165.650, Y  +453.156, Z    +0.000, E1   +30.934, E3 +440806.853}
SPL {X  -165.650, Y  +450.433, Z    +0.000, E1   +30.789, E3 +440817.209}
SPL {X  -165.650, Y  +447.097, Z    +0.000, E1   +30.843, E3 +440828.257}
SPL {X  -165.650, Y  +443.673, Z    +0.000, E1   +30.907, E3 +440839.565}
SPL {X  -165.650, Y  +439.486, Z    +0.000, E1   +30.857, E3 +440854.374}
SPL {X  -165.650, Y  +435.146, Z    +0.000, E1   +30.969, E3 +440868.293}
SPL {X  -165.650, Y  +431.607, Z    +0.000, E1   +30.889, E3 +440881.008}
SPL {X  -165.650, Y  +427.340, Z    +0.000, E1   +30.870, E3 +440895.720}
SPL {X  -165.650, Y  +423.901, Z    +0.000, E1   +30.858, E3 +440907.476}
SPL {X  -165.650, Y  +421.437, Z    +0.000, E1   +30.833, E3 +440916.074}
SPL {X  -165.650, Y  +418.489, Z    +0.000, E1   +30.835, E3 +440926.191}
SPL {X  -165.650, Y  +414.127, Z    +0.000, E1   +30.869, E3 +440941.100}
SPL {X  -165.650, Y  +408.547, Z    +0.000, E1   +30.964, E3 +440959.515}
SPL {X  -165.650, Y  +405.433, Z    +0.000, E1   +30.730, E3 +440971.492}
SPL {X  -165.650, Y  +401.473, Z    +0.000, E1   +30.933, E3 +440983.941}
SPL {X  -165.650, Y  +396.018, Z    +0.000, E1   +30.861, E3 +441003.126}
SPL {X  -165.650, Y  +391.522, Z    +0.000, E1   +30.837, E3 +441018.483}
SPL {X  -165.650, Y  +387.533, Z    +0.000, E1   +30.858, E3 +441032.109}
SPL {X  -165.650, Y  +383.627, Z    +0.000, E1   +30.885, E3 +441045.169}
SPL {X  -165.650, Y  +380.752, Z    +0.000, E1   +30.927, E3 +441054.683}
SPL {X  -165.648, Y  +377.739, Z    +0.000, E1   +30.835, E3 +441065.693}
SPL {X  -165.594, Y  +374.183, Z    +0.000, E1   +30.878, E3 +441077.529}
SPL {X  -165.429, Y  +369.945, Z    +0.000, E1   +30.850, E3 +441092.404}
SPL {X  -165.167, Y  +365.866, Z    +0.000, E1   +30.741, E3 +441106.937}
SPL {X  -164.892, Y  +362.671, Z    +0.000, E1   +30.830, E3 +441117.261}
SPL {X  -164.570, Y  +359.612, Z    +0.000, E1   +30.773, E3 +441128.074}
SPL {X  -164.104, Y  +355.923, Z    +0.000, E1   +30.626, E3 +441141.790}
SPL {X  -163.573, Y  +352.353, Z    +0.000, E1   +30.451, E3 +441155.055}
SPL {X  -162.976, Y  +348.856, Z    +0.000, E1   +30.757, E3 +441164.979}
SPL {X  -161.497, Y  +341.640, Z    +0.000, E1   +33.276, E3 +441172.256}
SPL {X  -152.976, Y  +314.952, Z    +0.000, E1   +38.607, E3 +441216.601}
SPL {X  -137.967, Y  +286.821, Z    +0.000, E1   +43.969, E3 +441259.822}
ENDSPLINE

SPLINE
SPL {X  -149.143, Y  +306.414, Z    +0.000, E1   +36.361, E3 +441310.954}
SPL {X  -164.268, Y  +357.145, Z    +0.000, E1   +15.880, E3 +441268.714}
SPL {X  -165.510, Y  +371.680, Z    +0.000, E1    +7.684, E3 +441271.716}
SPL {X  -165.628, Y  +375.818, Z    +0.000, E1    +5.016, E3 +441279.645}
SPL {X  -165.650, Y  +383.362, Z    +0.000, E1    +0.177, E3 +441260.679}
SPL {X  -165.650, Y  +383.923, Z    +0.000, E1    -0.215, E3 +441273.836}
SPL {X  -165.650, Y  +388.083, Z    +0.000, E1    -3.355, E3 +441272.700}
SPL {X  -165.650, Y  +395.510, Z    +0.000, E1    -9.810, E3 +441268.826}
SPL {X  -165.650, Y  +403.066, Z    +0.000, E1   -17.886, E3 +441261.659}
SPL {X  -165.650, Y  +416.345, Z    +0.000, E1   -29.511, E3 +441263.402}
SPL {X  -165.650, Y  +422.331, Z    +0.000, E1   -27.760, E3 +441288.901}
SPL {X  -165.650, Y  +441.276, Z    +0.000, E1   -37.343, E3 +441298.758}
SPL {X  -165.650, Y  +462.890, Z    +0.000, E1   -40.484, E3 +441332.841}
ENDSPLINE

SPLINE
SPL {X  -165.650, Y  +446.920, Z    +0.000, E1   -31.238, E3 +441345.167}
ENDSPLINE

SPLINE
SPL {X  -165.650, Y  +447.935, Z    +0.000, E1   -30.213, E3 +441355.455}
SPL {X  -165.650, Y  +451.020, Z    +0.000, E1   -30.224, E3 +441366.275}
SPL {X  -165.650, Y  +454.519, Z    +0.000, E1   -30.374, E3 +441377.457}
SPL {X  -165.650, Y  +457.429, Z    +0.000, E1   -30.029, E3 +441390.159}
SPL {X  -165.650, Y  +461.678, Z    +0.000, E1   -30.426, E3 +441402.284}
SPL {X  -165.650, Y  +463.853, Z    +0.000, E1   -30.103, E3 +441412.123}
SPL {X  -165.650, Y  +468.397, Z    +0.000, E1   -30.302, E3 +441426.927}
SPL {X  -165.650, Y  +472.566, Z    +0.000, E1   -30.124, E3 +441442.636}
SPL {X  -165.650, Y  +475.265, Z    +0.000, E1   -30.034, E3 +441452.674}
SPL {X  -165.650, Y  +477.862, Z    +0.000, E1   -30.319, E3 +441459.866}
SPL {X  -165.650, Y  +481.042, Z    +0.000, E1   -30.192, E3 +441472.126}
SPL {X  -165.650, Y  +485.236, Z    +0.000, E1   -30.294, E3 +441485.981}
SPL {X  -165.650, Y  +488.041, Z    +0.000, E1   -30.253, E3 +441496.103}
SPL {X  -165.650, Y  +491.281, Z    +0.000, E1   -30.148, E3 +441508.241}
SPL {X  -165.650, Y  +495.051, Z    +0.000, E1   -30.213, E3 +441521.049}
SPL {X  -165.650, Y  +499.546, Z    +0.000, E1   -30.283, E3 +441536.492}
SPL {X  -165.650, Y  +503.544, Z    +0.000, E1   -30.247, E3 +441550.561}
SPL {X  -165.650, Y  +506.344, Z    +0.000, E1   -30.129, E3 +441561.229}
SPL {X  -165.650, Y  +510.660, Z    +0.000, E1   -30.223, E3 +441575.933}
SPL {X  -165.650, Y  +514.670, Z    +0.000, E1   -30.278, E3 +441589.443}
SPL {X  -165.650, Y  +517.919, Z    +0.000, E1   -30.227, E3 +441601.302}
SPL {X  -165.650, Y  +522.822, Z    +0.000, E1   -30.289, E3 +441618.191}
SPL {X  -165.650, Y  +527.393, Z    +0.000, E1   -30.104, E3 +441635.439}
SPL {X  -165.650, Y  +531.783, Z    +0.000, E1   -30.416, E3 +441648.617}
SPL {X  -165.650, Y  +534.115, Z    +0.000, E1   -30.089, E3 +441658.999}
SPL {X  -165.650, Y  +537.522, Z    +0.000, E1   -30.251, E3 +441669.913}
SPL {X  -165.650, Y  +540.621, Z    +0.000, E1   -30.014, E3 +441682.474}
SPL {X  -165.650, Y  +544.944, Z    +0.000, E1   -30.447, E3 +441694.674}
SPL {X  -165.650, Y  +547.199, Z    +0.000, E1   -30.132, E3 +441704.647}
SPL {X  -165.650, Y  +550.512, Z    +0.000, E1   -30.197, E3 +441715.973}
SPL {X  -165.650, Y  +553.852, Z    +0.000, E1   -30.156, E3 +441727.914}
SPL {X  -165.650, Y  +557.277, Z    +0.000, E1   -30.150, E3 +441740.088}
SPL {X  -165.650, Y  +561.168, Z    +0.000, E1   -30.194, E3 +441753.470}
SPL {X  -165.650, Y  +565.528, Z    +0.000, E1   -30.192, E3 +441768.953}
SPL {X  -165.650, Y  +570.048, Z    +0.000, E1   -30.238, E3 +441784.384}
SPL {X  -165.650, Y  +573.110, Z    +0.000, E1   -30.057, E3 +441796.369}
SPL {X  -165.650, Y  +577.587, Z    +0.000, E1   -30.270, E3 +441810.808}
SPL {X  -165.650, Y  +581.190, Z    +0.000, E1   -30.107, E3 +441824.447}
SPL {X  -165.650, Y  +585.053, Z    +0.000, E1   -30.090, E3 +441838.317}
ENDSPLINE

SPLINE
SPL {X  -165.650, Y  +484.445, Z    +0.000, E1   +32.277, E3 +441855.722}
SPL {X  -165.650, Y  +481.524, Z    +0.000, E1   +31.089, E3 +441873.172}
SPL {X  -165.650, Y  +478.014, Z    +0.000, E1   +30.826, E3 +441886.780}
SPL {X  -165.650, Y  +474.473, Z    +0.000, E1   +30.943, E3 +441898.104}
SPL {X  -165.650, Y  +471.826, Z    +0.000, E1   +30.770, E3 +441908.288}
SPL {X  -165.650, Y  +467.753, Z    +0.000, E1   +30.878, E3 +441921.661}
SPL {X  -165.650, Y  +463.837, Z    +0.000, E1   +30.924, E3 +441934.595}
SPL {X  -165.650, Y  +461.106, Z    +0.000, E1   +30.916, E3 +441943.982}
SPL {X  -165.650, Y  +457.156, Z    +0.000, E1   +30.860, E3 +441958.058}
SPL {X  -165.650, Y  +453.156, Z    +0.000, E1   +30.934, E3 +441971.032}
SPL {X  -165.650, Y  +450.433, Z    +0.000, E1   +30.789, E3 +441981.388}
SPL {X  -165.650, Y  +447.097, Z    +0.000, E1   +30.843, E3 +441992.436}
SPL {X  -165.650, Y  +443.673, Z    +0.000, E1   +30.907, E3 +442003.744}
SPL {X  -165.650, Y  +439.486, Z    +0.000, E1   +30.857, E3 +442018.553}
SPL {X  -165.650, Y  +435.146, Z    +0.000, E1   +30.969, E3 +442032.473}
SPL {X  -165.650, Y  +431.607, Z    +0.000, E1   +30.889, E3 +442045.187}
SPL {X  -165.650, Y  +427.340, Z    +0.000, E1   +30.870, E3 +442059.899}
SPL {X  -165.650, Y  +423.901, Z    +0.000, E1   +30.858, E3 +442071.655}
SPL {X  -165.650, Y  +421.437, Z    +0.000, E1   +30.833, E3 +442080.253}
SPL {X  -165.650, Y  +418.489, Z    +0.000, E1   +30.835, E3 +442090.370}
SPL {X  -165.650, Y  +414.127, Z    +0.000, E1   +30.869, E3 +442105.279}
SPL {X  -165.650, Y  +408.547, Z    +0.000, E1   +30.964, E3 +442123.694}
SPL {X  -165.650, Y  +405.433, Z    +0.000, E1   +30.730, E3 +442135.671}
SPL {X  -165.650, Y  +401.473, Z    +0.000, E1   +30.933, E3 +442148.120}
SPL {X  -165.650, Y  +396.018, Z    +0.000, E1   +30.861, E3 +442167.305}
SPL {X  -165.650, Y  +390.331, Z    +0.000, E1   +30.892, E3 +442186.557}
SPL {X  -165.650, Y  +384.849, Z    +0.000, E1   +30.885, E3 +442205.360}
SPL {X  -165.650, Y  +380.752, Z    +0.000, E1   +30.927, E3 +442218.862}
SPL {X  -165.648, Y  +377.739, Z    +0.000, E1   +30.835, E3 +442229.872}
SPL {X  -165.594, Y  +374.183, Z    +0.000, E1   +30.878, E3 +442241.708}
SPL {X  -165.492, Y  +371.263, Z    +0.000, E1   +30.913, E3 +442251.403}
SPL {X  -165.379, Y  +369.027, Z    +0.000, E1   +30.727, E3 +442260.342}
SPL {X  -165.167, Y  +365.866, Z    +0.000, E1   +30.741, E3 +442271.116}
SPL {X  -164.892, Y  +362.671, Z    +0.000, E1   +30.830, E3 +442281.440}
SPL {X  -164.570, Y  +359.612, Z    +0.000, E1   +30.773, E3 +442292.253}
SPL {X  -164.104, Y  +355.923, Z    +0.000, E1   +30.626, E3 +442305.969}
SPL {X  -163.573, Y  +352.353, Z    +0.000, E1   +30.451, E3 +442319.234}
SPL {X  -162.476, Y  +346.230, Z    +0.000, E1   +31.677, E3 +442331.815}
SPL {X  -152.976, Y  +314.952, Z    +0.000, E1   +38.607, E3 +442380.780}
SPL {X  -137.967, Y  +286.821, Z    +0.000, E1   +43.969, E3 +442424.001}
ENDSPLINE

SPLINE
SPL {X  -153.316, Y  +315.777, Z    +0.000, E1   +33.140, E3 +442466.629}
SPL {X  -164.446, Y  +358.564, Z    +0.000, E1   +15.149, E3 +442431.839}
SPL {X  -165.379, Y  +369.025, Z    +0.000, E1    +9.158, E3 +442437.564}
SPL {X  -165.612, Y  +374.969, Z    +0.000, E1    +5.630, E3 +442440.240}
SPL {X  -165.650, Y  +383.362, Z    +0.000, E1    +0.177, E3 +442424.858}
SPL {X  -165.650, Y  +383.923, Z    +0.000, E1    -0.215, E3 +442438.015}
SPL {X  -165.650, Y  +388.083, Z    +0.000, E1    -3.355, E3 +442436.879}
SPL {X  -165.650, Y  +393.983, Z    +0.000, E1    -8.501, E3 +442433.277}
SPL {X  -165.650, Y  +402.241, Z    +0.000, E1   -16.711, E3 +442427.789}
SPL {X  -165.650, Y  +416.345, Z    +0.000, E1   -29.511, E3 +442427.581}
SPL {X  -165.650, Y  +422.331, Z    +0.000, E1   -27.760, E3 +442453.080}
SPL {X  -165.650, Y  +441.276, Z    +0.000, E1   -37.343, E3 +442462.937}
SPL {X  -165.650, Y  +462.890, Z    +0.000, E1   -40.484, E3 +442497.020}
ENDSPLINE

SPLINE
SPL {X  -165.650, Y  +446.920, Z    +0.000, E1   -31.238, E3 +442509.346}
ENDSPLINE

SPLINE
SPL {X  -165.650, Y  +447.935, Z    +0.000, E1   -30.213, E3 +442519.634}
SPL {X  -165.650, Y  +451.020, Z    +0.000, E1   -30.224, E3 +442530.454}
SPL {X  -165.650, Y  +454.519, Z    +0.000, E1   -30.374, E3 +442541.636}
SPL {X  -165.650, Y  +456.542, Z    +0.000, E1   -29.986, E3 +442551.381}
SPL {X  -165.650, Y  +460.618, Z    +0.000, E1   -30.298, E3 +442563.702}
SPL {X  -165.650, Y  +463.853, Z    +0.000, E1   -30.103, E3 +442576.302}
SPL {X  -165.650, Y  +467.246, Z    +0.000, E1   -30.279, E3 +442587.033}
SPL {X  -165.650, Y  +469.780, Z    +0.000, E1   -30.237, E3 +442596.158}
SPL {X  -165.650, Y  +472.566, Z    +0.000, E1   -30.124, E3 +442606.816}
SPL {X  -165.650, Y  +476.540, Z    +0.000, E1   -30.193, E3 +442620.360}
SPL {X  -165.650, Y  +480.320, Z    +0.000, E1   -30.163, E3 +442633.837}
SPL {X  -165.650, Y  +484.477, Z    +0.000, E1   -30.274, E3 +442647.727}
SPL {X  -165.650, Y  +488.041, Z    +0.000, E1   -30.253, E3 +442660.282}
SPL {X  -165.650, Y  +491.281, Z    +0.000, E1   -30.148, E3 +442672.420}
SPL {X  -165.650, Y  +495.051, Z    +0.000, E1   -30.213, E3 +442685.229}
SPL {X  -165.650, Y  +498.418, Z    +0.000, E1   -30.282, E3 +442696.521}
SPL {X  -165.650, Y  +500.833, Z    +0.000, E1   -30.191, E3 +442705.571}
SPL {X  -165.650, Y  +504.246, Z    +0.000, E1   -30.231, E3 +442717.437}
SPL {X  -165.650, Y  +507.017, Z    +0.000, E1   -30.108, E3 +442727.845}
SPL {X  -165.650, Y  +510.660, Z    +0.000, E1   -30.223, E3 +442740.112}
SPL {X  -165.650, Y  +515.918, Z    +0.000, E1   -30.316, E3 +442757.920}
SPL {X  -165.650, Y  +520.621, Z    +0.000, E1   -30.198, E3 +442775.205}
SPL {X  -165.650, Y  +525.344, Z    +0.000, E1   -30.269, E3 +442791.262}
SPL {X  -165.650, Y  +528.152, Z    +0.000, E1   -29.991, E3 +442802.903}
SPL {X  -165.650, Y  +531.783, Z    +0.000, E1   -30.416, E3 +442812.796}
SPL {X  -165.650, Y  +534.115, Z    +0.000, E1   -30.089, E3 +442823.178}
SPL {X  -165.650, Y  +538.363, Z    +0.000, E1   -30.232, E3 +442837.348}
SPL {X  -165.650, Y  +543.650, Z    +0.000, E1   -30.281, E3 +442855.567}
SPL {X  -165.650, Y  +547.199, Z    +0.000, E1   -30.132, E3 +442868.826}
SPL {X  -165.650, Y  +550.512, Z    +0.000, E1   -30.197, E3 +442880.152}
SPL {X  -165.650, Y  +554.908, Z    +0.000, E1   -30.180, E3 +442895.813}
SPL {X  -165.650, Y  +560.243, Z    +0.000, E1   -30.214, E3 +442914.439}
SPL {X  -165.650, Y  +565.528, Z    +0.000, E1   -30.192, E3 +442933.132}
SPL {X  -165.650, Y  +570.048, Z    +0.000, E1   -30.238, E3 +442948.563}
SPL {X  -165.650, Y  +573.110, Z    +0.000, E1   -30.057, E3 +442960.548}
SPL {X  -165.650, Y  +577.587, Z    +0.000, E1   -30.270, E3 +442974.987}
SPL {X  -165.650, Y  +581.190, Z    +0.000, E1   -30.107, E3 +442988.626}
SPL {X  -165.650, Y  +585.053, Z    +0.000, E1   -30.090, E3 +443002.496}
ENDSPLINE

SPLINE
SPL {X  -165.650, Y  +484.445, Z    +0.000, E1   +32.277, E3 +443019.901}
SPL {X  -165.650, Y  +481.524, Z    +0.000, E1   +31.089, E3 +443037.351}
SPL {X  -165.650, Y  +478.014, Z    +0.000, E1   +30.826, E3 +443050.959}
SPL {X  -165.650, Y  +474.473, Z    +0.000, E1   +30.943, E3 +443062.283}
SPL {X  -165.650, Y  +471.826, Z    +0.000, E1   +30.770, E3 +443072.467}
SPL {X  -165.650, Y  +467.753, Z    +0.000, E1   +30.878, E3 +443085.840}
SPL {X  -165.650, Y  +463.837, Z    +0.000, E1   +30.924, E3 +443098.774}
SPL {X  -165.650, Y  +461.106, Z    +0.000, E1   +30.916, E3 +443108.161}
SPL {X  -165.650, Y  +457.156, Z    +0.000, E1   +30.860, E3 +443122.238}
SPL {X  -165.650, Y  +453.156, Z    +0.000, E1   +30.934, E3 +443135.211}
SPL {X  -165.650, Y  +450.433, Z    +0.000, E1   +30.789, E3 +443145.567}
SPL {X  -165.650, Y  +447.097, Z    +0.000, E1   +30.843, E3 +443156.615}
SPL {X  -165.650, Y  +443.673, Z    +0.000, E1   +30.907, E3 +443167.923}
SPL {X  -165.650, Y  +439.486, Z    +0.000, E1   +30.857, E3 +443182.732}
SPL {X  -165.650, Y  +435.146, Z    +0.000, E1   +30.969, E3 +443196.652}
SPL {X  -165.650, Y  +431.607, Z    +0.000, E1   +30.889, E3 +443209.366}
SPL {X  -165.650, Y  +427.340, Z    +0.000, E1   +30.870, E3 +443224.078}
SPL {X  -165.650, Y  +423.901, Z    +0.000, E1   +30.858, E3 +443235.834}
SPL {X  -165.650, Y  +421.437, Z    +0.000, E1   +30.833, E3 +443244.432}
SPL {X  -165.650, Y  +418.489, Z    +0.000, E1   +30.835, E3 +443254.549}
SPL {X  -165.650, Y  +414.127, Z    +0.000, E1   +30.869, E3 +443269.458}
SPL {X  -165.650, Y  +408.547, Z    +0.000, E1   +30.964, E3 +443287.873}
SPL {X  -165.650, Y  +405.433, Z    +0.000, E1   +30.730, E3 +443299.850}
SPL {X  -165.650, Y  +401.473, Z    +0.000, E1   +30.933, E3 +443312.299}
SPL {X  -165.650, Y  +396.018, Z    +0.000, E1   +30.861, E3 +443331.484}
SPL {X  -165.650, Y  +390.331, Z    +0.000, E1   +30.892, E3 +443350.736}
SPL {X  -165.650, Y  +384.849, Z    +0.000, E1   +30.885, E3 +443369.539}
SPL {X  -165.650, Y  +380.752, Z    +0.000, E1   +30.927, E3 +443383.041}
SPL {X  -165.648, Y  +377.739, Z    +0.000, E1   +30.835, E3 +443394.051}
SPL {X  -165.594, Y  +374.183, Z    +0.000, E1   +30.878, E3 +443405.888}
SPL {X  -165.492, Y  +371.263, Z    +0.000, E1   +30.913, E3 +443415.583}
SPL {X  -165.379, Y  +369.027, Z    +0.000, E1   +30.727, E3 +443424.521}
SPL {X  -165.167, Y  +365.866, Z    +0.000, E1   +30.741, E3 +443435.295}
SPL {X  -164.892, Y  +362.671, Z    +0.000, E1   +30.830, E3 +443445.619}
SPL {X  -164.570, Y  +359.612, Z    +0.000, E1   +30.773, E3 +443456.432}
SPL {X  -164.104, Y  +355.923, Z    +0.000, E1   +30.626, E3 +443470.148}
SPL {X  -163.573, Y  +352.353, Z    +0.000, E1   +30.451, E3 +443483.413}
SPL {X  -162.476, Y  +346.230, Z    +0.000, E1   +31.677, E3 +443495.994}
SPL {X  -152.976, Y  +314.952, Z    +0.000, E1   +38.607, E3 +443544.959}
SPL {X  -137.967, Y  +286.821, Z    +0.000, E1   +43.969, E3 +443588.180}
ENDSPLINE

SPLINE
SPL {X  -153.316, Y  +315.777, Z    +0.000, E1   +33.140, E3 +443630.808}
SPL {X  -164.446, Y  +358.564, Z    +0.000, E1   +15.149, E3 +443596.019}
SPL {X  -165.510, Y  +371.680, Z    +0.000, E1    +7.684, E3 +443600.074}
SPL {X  -165.628, Y  +375.818, Z    +0.000, E1    +5.016, E3 +443608.004}
SPL {X  -165.650, Y  +383.362, Z    +0.000, E1    +0.177, E3 +443589.037}
SPL {X  -165.650, Y  +383.923, Z    +0.000, E1    -0.215, E3 +443602.195}
SPL {X  -165.650, Y  +388.083, Z    +0.000, E1    -3.355, E3 +443601.058}
SPL {X  -165.650, Y  +393.983, Z    +0.000, E1    -8.501, E3 +443597.456}
SPL {X  -165.650, Y  +402.241, Z    +0.000, E1   -16.711, E3 +443591.968}
SPL {X  -165.650, Y  +416.345, Z    +0.000, E1   -29.511, E3 +443591.760}
SPL {X  -165.650, Y  +422.331, Z    +0.000, E1   -27.760, E3 +443617.259}
SPL {X  -165.650, Y  +441.276, Z    +0.000, E1   -37.343, E3 +443627.116}
SPL {X  -165.650, Y  +462.890, Z    +0.000, E1   -40.484, E3 +443661.199}
ENDSPLINE

SPLINE
SPL {X  -165.650, Y  +446.920, Z    +0.000, E1   -31.238, E3 +443673.525}
ENDSPLINE

SPLINE
SPL {X  -165.650, Y  +447.935, Z    +0.000, E1   -30.213, E3 +443683.813}
SPL {X  -165.650, Y  +451.020, Z    +0.000, E1   -30.224, E3 +443694.633}
SPL {X  -165.650, Y  +454.519, Z    +0.000, E1   -30.374, E3 +443705.816}
SPL {X  -165.650, Y  +456.542, Z    +0.000, E1   -29.986, E3 +443715.560}
SPL {X  -165.650, Y  +460.618, Z    +0.000, E1   -30.298, E3 +443727.881}
SPL {X  -165.650, Y  +463.853, Z    +0.000, E1   -30.103, E3 +443740.482}
SPL {X  -165.650, Y  +468.397, Z    +0.000, E1   -30.302, E3 +443755.285}
SPL {X  -165.650, Y  +472.566, Z    +0.000, E1   -30.124, E3 +443770.995}
SPL {X  -165.650, Y  +475.265, Z    +0.000, E1   -30.034, E3 +443781.032}
SPL {X  -165.650, Y  +477.862, Z    +0.000, E1   -30.319, E3 +443788.224}
SPL {X  -165.650, Y  +481.042, Z    +0.000, E1   -30.192, E3 +443800.484}
SPL {X  -165.650, Y  +485.236, Z    +0.000, E1   -30.294, E3 +443814.340}
SPL {X  -165.650, Y  +488.041, Z    +0.000, E1   -30.253, E3 +443824.461}
SPL {X  -165.650, Y  +491.281, Z    +0.000, E1   -30.148, E3 +443836.599}
SPL {X  -165.650, Y  +495.051, Z    +0.000, E1   -30.213, E3 +443849.408}
SPL {X  -165.650, Y  +499.546, Z    +0.000, E1   -30.283, E3 +443864.851}
SPL {X  -165.650, Y  +503.544, Z    +0.000, E1   -30.247, E3 +443878.919}
SPL {X  -165.650, Y  +506.344, Z    +0.000, E1   -30.129, E3 +443889.588}
SPL {X  -165.650, Y  +510.660, Z    +0.000, E1   -30.223, E3 +443904.291}
SPL {X  -165.650, Y  +514.670, Z    +0.000, E1   -30.278, E3 +443917.801}
SPL {X  -165.650, Y  +517.919, Z    +0.000, E1   -30.227, E3 +443929.660}
SPL {X  -165.650, Y  +521.521, Z    +0.000, E1   -30.210, E3 +443942.335}
SPL {X  -165.650, Y  +525.344, Z    +0.000, E1   -30.269, E3 +443955.441}
SPL {X  -165.650, Y  +528.152, Z    +0.000, E1   -29.991, E3 +443967.082}
SPL {X  -165.650, Y  +531.783, Z    +0.000, E1   -30.416, E3 +443976.975}
SPL {X  -165.650, Y  +534.115, Z    +0.000, E1   -30.089, E3 +443987.357}
SPL {X  -165.650, Y  +537.522, Z    +0.000, E1   -30.251, E3 +443998.271}
SPL {X  -165.650, Y  +540.621, Z    +0.000, E1   -30.014, E3 +444010.832}
SPL {X  -165.650, Y  +544.944, Z    +0.000, E1   -30.447, E3 +444023.032}
SPL {X  -165.650, Y  +548.549, Z    +0.000, E1   -30.216, E3 +444037.355}
SPL {X  -165.650, Y  +553.092, Z    +0.000, E1   -30.157, E3 +444053.698}
SPL {X  -165.650, Y  +557.277, Z    +0.000, E1   -30.150, E3 +444068.446}
SPL {X  -165.650, Y  +561.168, Z    +0.000, E1   -30.194, E3 +444081.828}
SPL {X  -165.650, Y  +564.449, Z    +0.000, E1   -30.167, E3 +444093.511}
SPL {X  -165.650, Y  +566.935, Z    +0.000, E1   -30.135, E3 +444102.417}
SPL {X  -165.650, Y  +570.048, Z    +0.000, E1   -30.238, E3 +444112.742}
SPL {X  -165.650, Y  +573.110, Z    +0.000, E1   -30.057, E3 +444124.727}
SPL {X  -165.650, Y  +576.497, Z    +0.000, E1   -30.234, E3 +444135.425}
SPL {X  -165.650, Y  +580.354, Z    +0.000, E1   -30.196, E3 +444149.440}
SPL {X  -165.650, Y  +585.053, Z    +0.000, E1   -30.090, E3 +444166.675}
ENDSPLINE

SPLINE
SPL {X  -165.650, Y  +484.445, Z    +0.000, E1   +32.277, E3 +444184.080}
SPL {X  -165.650, Y  +481.524, Z    +0.000, E1   +31.089, E3 +444201.530}
SPL {X  -165.650, Y  +478.014, Z    +0.000, E1   +30.826, E3 +444215.138}
SPL {X  -165.650, Y  +474.473, Z    +0.000, E1   +30.943, E3 +444226.462}
SPL {X  -165.650, Y  +470.376, Z    +0.000, E1   +30.888, E3 +444240.992}
SPL {X  -165.650, Y  +465.146, Z    +0.000, E1   +30.883, E3 +444258.922}
SPL {X  -165.650, Y  +461.106, Z    +0.000, E1   +30.916, E3 +444272.340}
SPL {X  -165.650, Y  +458.435, Z    +0.000, E1   +30.759, E3 +444282.548}
SPL {X  -165.650, Y  +454.220, Z    +0.000, E1   +30.954, E3 +444295.781}
SPL {X  -165.650, Y  +450.433, Z    +0.000, E1   +30.789, E3 +444309.746}
SPL {X  -165.650, Y  +447.097, Z    +0.000, E1   +30.843, E3 +444320.795}
SPL {X  -165.650, Y  +443.673, Z    +0.000, E1   +30.907, E3 +444332.102}
SPL {X  -165.650, Y  +440.976, Z    +0.000, E1   +30.719, E3 +444342.559}
SPL {X  -165.650, Y  +437.973, Z    +0.000, E1   +30.928, E3 +444351.431}
SPL {X  -165.650, Y  +434.043, Z    +0.000, E1   +30.950, E3 +444364.927}
SPL {X  -165.650, Y  +430.419, Z    +0.000, E1   +30.895, E3 +444377.430}
SPL {X  -165.650, Y  +427.340, Z    +0.000, E1   +30.870, E3 +444388.257}
SPL {X  -165.650, Y  +422.641, Z    +0.000, E1   +30.884, E3 +444404.346}
SPL {X  -165.650, Y  +418.489, Z    +0.000, E1   +30.835, E3 +444418.728}
SPL {X  -165.650, Y  +414.127, Z    +0.000, E1   +30.869, E3 +444433.637}
SPL {X  -165.650, Y  +408.547, Z    +0.000, E1   +30.964, E3 +444452.052}
SPL {X  -165.650, Y  +405.433, Z    +0.000, E1   +30.730, E3 +444464.030}
SPL {X  -165.650, Y  +402.516, Z    +0.000, E1   +30.874, E3 +444473.152}
SPL {X  -165.650, Y  +398.147, Z    +0.000, E1   +30.902, E3 +444488.031}
SPL {X  -165.650, Y  +394.694, Z    +0.000, E1   +30.805, E3 +444500.339}
SPL {X  -165.650, Y  +391.522, Z    +0.000, E1   +30.837, E3 +444511.020}
SPL {X  -165.650, Y  +387.533, Z    +0.000, E1   +30.858, E3 +444524.646}
SPL {X  -165.650, Y  +383.627, Z    +0.000, E1   +30.885, E3 +444537.706}
SPL {X  -165.650, Y  +379.886, Z    +0.000, E1   +30.887, E3 +444550.595}
SPL {X  -165.614, Y  +375.058, Z    +0.000, E1   +30.905, E3 +444567.048}
SPL {X  -165.492, Y  +371.263, Z    +0.000, E1   +30.913, E3 +444579.762}
SPL {X  -165.379, Y  +369.027, Z    +0.000, E1   +30.727, E3 +444588.700}
SPL {X  -165.167, Y  +365.866, Z    +0.000, E1   +30.741, E3 +444599.474}
SPL {X  -164.892, Y  +362.671, Z    +0.000, E1   +30.830, E3 +444609.798}
SPL {X  -164.570, Y  +359.612, Z    +0.000, E1   +30.773, E3 +444620.611}
SPL {X  -164.104, Y  +355.923, Z    +0.000, E1   +30.626, E3 +444634.327}
SPL {X  -163.573, Y  +352.353, Z    +0.000, E1   +30.451, E3 +444647.592}
SPL {X  -162.976, Y  +348.856, Z    +0.000, E1   +30.757, E3 +444657.516}
SPL {X  -161.497, Y  +341.640, Z    +0.000, E1   +33.276, E3 +444664.794}
SPL {X  -152.976, Y  +314.952, Z    +0.000, E1   +38.607, E3 +444709.138}
SPL {X  -137.967, Y  +286.821, Z    +0.000, E1   +43.969, E3 +444752.359}
ENDSPLINE

SPLINE
SPL {X  -149.143, Y  +306.414, Z    +0.000, E1   +36.361, E3 +444803.492}
SPL {X  -164.268, Y  +357.145, Z    +0.000, E1   +15.880, E3 +444761.251}
SPL {X  -165.379, Y  +369.025, Z    +0.000, E1    +9.158, E3 +444765.922}
SPL {X  -165.612, Y  +374.969, Z    +0.000, E1    +5.630, E3 +444768.598}
SPL {X  -165.650, Y  +383.362, Z    +0.000, E1    +0.177, E3 +444753.216}
SPL {X  -165.650, Y  +383.923, Z    +0.000, E1    -0.215, E3 +444766.374}
SPL {X  -165.650, Y  +388.083, Z    +0.000, E1    -3.355, E3 +444765.237}
SPL {X  -165.650, Y  +393.983, Z    +0.000, E1    -8.501, E3 +444761.635}
SPL {X  -165.650, Y  +402.241, Z    +0.000, E1   -16.711, E3 +444756.147}
SPL {X  -165.650, Y  +416.345, Z    +0.000, E1   -29.511, E3 +444755.939}
SPL {X  -165.650, Y  +422.331, Z    +0.000, E1   -27.760, E3 +444781.438}
SPL {X  -165.650, Y  +441.276, Z    +0.000, E1   -37.343, E3 +444791.295}
SPL {X  -165.650, Y  +462.890, Z    +0.000, E1   -40.484, E3 +444825.378}
ENDSPLINE

SPLINE
SPL {X  -165.650, Y  +446.920, Z    +0.000, E1   -31.238, E3 +444837.704}
ENDSPLINE

SPLINE
SPL {X  -165.650, Y  +447.935, Z    +0.000, E1   -30.213, E3 +444847.992}
SPL {X  -165.650, Y  +451.020, Z    +0.000, E1   -30.224, E3 +444858.812}
SPL {X  -165.650, Y  +454.519, Z    +0.000, E1   -30.374, E3 +444869.995}
SPL {X  -165.650, Y  +456.542, Z    +0.000, E1   -29.986, E3 +444879.739}
SPL {X  -165.650, Y  +460.618, Z    +0.000, E1   -30.298, E3 +444892.060}
SPL {X  -165.650, Y  +463.853, Z    +0.000, E1   -30.103, E3 +444904.661}
SPL {X  -165.650, Y  +467.246, Z    +0.000, E1   -30.279, E3 +444915.391}
SPL {X  -165.650, Y  +469.780, Z    +0.000, E1   -30.237, E3 +444924.516}
SPL {X  -165.650, Y  +472.566, Z    +0.000, E1   -30.124, E3 +444935.174}
SPL {X  -165.650, Y  +476.540, Z    +0.000, E1   -30.193, E3 +444948.718}
SPL {X  -165.650, Y  +480.320, Z    +0.000, E1   -30.163, E3 +444962.196}
SPL {X  -165.650, Y  +484.477, Z    +0.000, E1   -30.274, E3 +444976.085}
SPL {X  -165.650, Y  +488.041, Z    +0.000, E1   -30.253, E3 +444988.640}
SPL {X  -165.650, Y  +491.281, Z    +0.000, E1   -30.148, E3 +445000.778}
SPL {X  -165.650, Y  +495.051, Z    +0.000, E1   -30.213, E3 +445013.587}
SPL {X  -165.650, Y  +498.418, Z    +0.000, E1   -30.282, E3 +445024.880}
SPL {X  -165.650, Y  +500.833, Z    +0.000, E1   -30.191, E3 +445033.929}
SPL {X  -165.650, Y  +504.246, Z    +0.000, E1   -30.231, E3 +445045.795}
SPL {X  -165.650, Y  +507.017, Z    +0.000, E1   -30.108, E3 +445056.203}
SPL {X  -165.650, Y  +510.660, Z    +0.000, E1   -30.223, E3 +445068.470}
SPL {X  -165.650, Y  +514.670, Z    +0.000, E1   -30.278, E3 +445081.980}
SPL {X  -165.650, Y  +517.919, Z    +0.000, E1   -30.227, E3 +445093.839}
SPL {X  -165.650, Y  +521.521, Z    +0.000, E1   -30.210, E3 +445106.514}
SPL {X  -165.650, Y  +525.344, Z    +0.000, E1   -30.269, E3 +445119.620}
SPL {X  -165.650, Y  +528.152, Z    +0.000, E1   -29.991, E3 +445131.261}
SPL {X  -165.650, Y  +531.783, Z    +0.000, E1   -30.416, E3 +445141.154}
SPL {X  -165.650, Y  +534.115, Z    +0.000, E1   -30.089, E3 +445151.536}
SPL {X  -165.650, Y  +538.363, Z    +0.000, E1   -30.232, E3 +445165.706}
SPL {X  -165.650, Y  +543.650, Z    +0.000, E1   -30.281, E3 +445183.926}
SPL {X  -165.650, Y  +547.199, Z    +0.000, E1   -30.132, E3 +445197.185}
SPL {X  -165.650, Y  +550.512, Z    +0.000, E1   -30.197, E3 +445208.510}
SPL {X  -165.650, Y  +553.852, Z    +0.000, E1   -30.156, E3 +445220.451}
SPL {X  -165.650, Y  +557.277, Z    +0.000, E1   -30.150, E3 +445232.626}
SPL {X  -165.650, Y  +561.168, Z    +0.000, E1   -30.194, E3 +445246.007}
SPL {X  -165.650, Y  +565.528, Z    +0.000, E1   -30.192, E3 +445261.490}
SPL {X  -165.650, Y  +570.048, Z    +0.000, E1   -30.238, E3 +445276.921}
SPL {X  -165.650, Y  +573.110, Z    +0.000, E1   -30.057, E3 +445288.906}
SPL {X  -165.650, Y  +577.587, Z    +0.000, E1   -30.270, E3 +445303.345}
SPL {X  -165.650, Y  +581.190, Z    +0.000, E1   -30.107, E3 +445316.984}
SPL {X  -165.650, Y  +585.053, Z    +0.000, E1   -30.090, E3 +445330.854}
ENDSPLINE

SPLINE
SPL {X  -165.650, Y  +484.968, Z    +0.000, E1   +32.508, E3 +445344.820}
SPL {X  -165.650, Y  +482.280, Z    +0.000, E1   +31.680, E3 +445359.147}
SPL {X  -165.650, Y  +479.331, Z    +0.000, E1   +30.680, E3 +445375.895}
SPL {X  -165.650, Y  +474.473, Z    +0.000, E1   +30.943, E3 +445390.641}
SPL {X  -165.650, Y  +471.826, Z    +0.000, E1   +30.770, E3 +445400.825}
SPL {X  -165.650, Y  +467.753, Z    +0.000, E1   +30.878, E3 +445414.198}
SPL {X  -165.650, Y  +463.837, Z    +0.000, E1   +30.924, E3 +445427.132}
SPL {X  -165.650, Y  +461.106, Z    +0.000, E1   +30.916, E3 +445436.519}
SPL {X  -165.650, Y  +458.435, Z    +0.000, E1   +30.759, E3 +445446.727}
SPL {X  -165.650, Y  +454.220, Z    +0.000, E1   +30.954, E3 +445459.960}
SPL {X  -165.650, Y  +450.433, Z    +0.000, E1   +30.789, E3 +445473.925}
SPL {X  -165.650, Y  +447.097, Z    +0.000, E1   +30.843, E3 +445484.974}
SPL {X  -165.650, Y  +443.673, Z    +0.000, E1   +30.907, E3 +445496.281}
SPL {X  -165.650, Y  +440.976, Z    +0.000, E1   +30.719, E3 +445506.738}
SPL {X  -165.650, Y  +437.973, Z    +0.000, E1   +30.928, E3 +445515.610}
SPL {X  -165.650, Y  +434.043, Z    +0.000, E1   +30.950, E3 +445529.107}
SPL {X  -165.650, Y  +430.419, Z    +0.000, E1   +30.895, E3 +445541.610}
SPL {X  -165.650, Y  +427.340, Z    +0.000, E1   +30.870, E3 +445552.436}
SPL {X  -165.650, Y  +422.641, Z    +0.000, E1   +30.884, E3 +445568.525}
SPL {X  -165.650, Y  +417.366, Z    +0.000, E1   +30.879, E3 +445586.631}
SPL {X  -165.650, Y  +413.181, Z    +0.000, E1   +30.815, E3 +445601.229}
SPL {X  -165.650, Y  +408.547, Z    +0.000, E1   +30.964, E3 +445616.232}
SPL {X  -165.650, Y  +403.421, Z    +0.000, E1   +30.863, E3 +445634.449}
SPL {X  -165.650, Y  +399.681, Z    +0.000, E1   +30.933, E3 +445646.532}
SPL {X  -165.650, Y  +396.018, Z    +0.000, E1   +30.861, E3 +445659.842}
SPL {X  -165.650, Y  +391.522, Z    +0.000, E1   +30.837, E3 +445675.199}
SPL {X  -165.650, Y  +387.533, Z    +0.000, E1   +30.858, E3 +445688.825}
SPL {X  -165.650, Y  +383.627, Z    +0.000, E1   +30.885, E3 +445701.886}
SPL {X  -165.650, Y  +380.752, Z    +0.000, E1   +30.927, E3 +445711.399}
SPL {X  -165.648, Y  +377.739, Z    +0.000, E1   +30.835, E3 +445722.409}
SPL {X  -165.594, Y  +374.183, Z    +0.000, E1   +30.878, E3 +445734.246}
SPL {X  -165.429, Y  +369.945, Z    +0.000, E1   +30.850, E3 +445749.121}
SPL {X  -165.167, Y  +365.866, Z    +0.000, E1   +30.741, E3 +445763.653}
SPL {X  -164.892, Y  +362.671, Z    +0.000, E1   +30.830, E3 +445773.977}
SPL {X  -164.570, Y  +359.612, Z    +0.000, E1   +30.773, E3 +445784.790}
SPL {X  -164.287, Y  +357.291, Z    +0.000, E1   +30.513, E3 +445794.419}
SPL {X  -163.720, Y  +353.284, Z    +0.000, E1   +30.592, E3 +445807.866}
SPL {X  -162.476, Y  +346.230, Z    +0.000, E1   +31.677, E3 +445824.352}
SPL {X  -152.976, Y  +314.952, Z    +0.000, E1   +38.607, E3 +445873.317}
SPL {X  -137.967, Y  +286.821, Z    +0.000, E1   +43.969, E3 +445916.538}
ENDSPLINE

SPLINE
SPL {X  -149.143, Y  +306.414, Z    +0.000, E1   +36.361, E3 +445967.671}
SPL {X  -163.091, Y  +349.496, Z    +0.000, E1   +19.699, E3 +445924.454}
SPL {X  -165.027, Y  +364.142, Z    +0.000, E1   +12.054, E3 +445927.594}
SPL {X  -165.612, Y  +374.969, Z    +0.000, E1    +5.630, E3 +445932.777}
SPL {X  -165.650, Y  +383.362, Z    +0.000, E1    +0.177, E3 +445917.395}
SPL {X  -165.650, Y  +383.923, Z    +0.000, E1    -0.215, E3 +445930.553}
SPL {X  -165.650, Y  +388.083, Z    +0.000, E1    -3.355, E3 +445929.416}
SPL {X  -165.650, Y  +393.983, Z    +0.000, E1    -8.501, E3 +445925.815}
SPL {X  -165.650, Y  +402.241, Z    +0.000, E1   -16.711, E3 +445920.326}
SPL {X  -165.650, Y  +416.345, Z    +0.000, E1   -29.511, E3 +445920.118}
SPL {X  -165.650, Y  +422.331, Z    +0.000, E1   -27.760, E3 +445945.617}
SPL {X  -165.650, Y  +441.276, Z    +0.000, E1   -37.343, E3 +445955.474}
SPL {X  -165.650, Y  +462.890, Z    +0.000, E1   -40.484, E3 +445989.557}
ENDSPLINE

SPLINE
SPL {X  -165.650, Y  +446.920, Z    +0.000, E1   -31.238, E3 +446001.883}
ENDSPLINE

SPLINE
SPL {X  -165.650, Y  +447.935, Z    +0.000, E1   -30.213, E3 +446012.171}
SPL {X  -165.650, Y  +451.020, Z    +0.000, E1   -30.224, E3 +446022.991}
SPL {X  -165.650, Y  +454.519, Z    +0.000, E1   -30.374, E3 +446034.174}
SPL {X  -165.650, Y  +457.429, Z    +0.000, E1   -30.029, E3 +446046.875}
SPL {X  -165.650, Y  +461.678, Z    +0.000, E1   -30.426, E3 +446059.000}
SPL {X  -165.650, Y  +463.853, Z    +0.000, E1   -30.103, E3 +446068.840}
SPL {X  -165.650, Y  +468.397, Z    +0.000, E1   -30.302, E3 +446083.644}
SPL {X  -165.650, Y  +472.566, Z    +0.000, E1   -30.124, E3 +446099.353}
SPL {X  -165.650, Y  +475.265, Z    +0.000, E1   -30.034, E3 +446109.390}
SPL {X  -165.650, Y  +477.862, Z    +0.000, E1   -30.319, E3 +446116.582}
SPL {X  -165.650, Y  +481.042, Z    +0.000, E1   -30.192, E3 +446128.842}
SPL {X  -165.650, Y  +485.236, Z    +0.000, E1   -30.294, E3 +446142.698}
SPL {X  -165.650, Y  +488.041, Z    +0.000, E1   -30.253, E3 +446152.819}
SPL {X  -165.650, Y  +491.281, Z    +0.000, E1   -30.148, E3 +446164.957}
SPL {X  -165.650, Y  +495.051, Z    +0.000, E1   -30.213, E3 +446177.766}
SPL {X  -165.650, Y  +498.418, Z    +0.000, E1   -30.282, E3 +446189.059}
SPL {X  -165.650, Y  +500.833, Z    +0.000, E1   -30.191, E3 +446198.108}
SPL {X  -165.650, Y  +504.246, Z    +0.000, E1   -30.231, E3 +446209.974}
SPL {X  -165.650, Y  +507.017, Z    +0.000, E1   -30.108, E3 +446220.383}
SPL {X  -165.650, Y  +510.660, Z    +0.000, E1   -30.223, E3 +446232.649}
SPL {X  -165.650, Y  +515.918, Z    +0.000, E1   -30.316, E3 +446250.457}
SPL {X  -165.650, Y  +520.621, Z    +0.000, E1   -30.198, E3 +446267.743}
SPL {X  -165.650, Y  +525.344, Z    +0.000, E1   -30.269, E3 +446283.799}
SPL {X  -165.650, Y  +528.152, Z    +0.000, E1   -29.991, E3 +446295.440}
SPL {X  -165.650, Y  +531.783, Z    +0.000, E1   -30.416, E3 +446305.333}
SPL {X  -165.650, Y  +534.115, Z    +0.000, E1   -30.089, E3 +446315.715}
SPL {X  -165.650, Y  +538.363, Z    +0.000, E1   -30.232, E3 +446329.885}
SPL {X  -165.650, Y  +543.650, Z    +0.000, E1   -30.281, E3 +446348.105}
SPL {X  -165.650, Y  +547.199, Z    +0.000, E1   -30.132, E3 +446361.364}
SPL {X  -165.650, Y  +550.512, Z    +0.000, E1   -30.197, E3 +446372.689}
SPL {X  -165.650, Y  +553.852, Z    +0.000, E1   -30.156, E3 +446384.630}
SPL {X  -165.650, Y  +557.277, Z    +0.000, E1   -30.150, E3 +446396.805}
SPL {X  -165.650, Y  +561.168, Z    +0.000, E1   -30.194, E3 +446410.186}
SPL {X  -165.650, Y  +564.449, Z    +0.000, E1   -30.167, E3 +446421.869}
SPL {X  -165.650, Y  +566.935, Z    +0.000, E1   -30.135, E3 +446430.775}
SPL {X  -165.650, Y  +570.048, Z    +0.000, E1   -30.238, E3 +446441.100}
SPL {X  -165.650, Y  +573.110, Z    +0.000, E1   -30.057, E3 +446453.085}
SPL {X  -165.650, Y  +576.497, Z    +0.000, E1   -30.234, E3 +446463.783}
SPL {X  -165.650, Y  +580.354, Z    +0.000, E1   -30.196, E3 +446477.798}
SPL {X  -165.650, Y  +585.053, Z    +0.000, E1   -30.090, E3 +446495.033}
ENDSPLINE

SPLINE
SPL {X  -165.650, Y  +484.445, Z    +0.000, E1   +32.277, E3 +446512.438}
SPL {X  -165.650, Y  +481.524, Z    +0.000, E1   +31.089, E3 +446529.889}
SPL {X  -165.650, Y  +478.014, Z    +0.000, E1   +30.826, E3 +446543.496}
SPL {X  -165.650, Y  +474.473, Z    +0.000, E1   +30.943, E3 +446554.821}
SPL {X  -165.650, Y  +470.376, Z    +0.000, E1   +30.888, E3 +446569.350}
SPL {X  -165.650, Y  +465.146, Z    +0.000, E1   +30.883, E3 +446587.280}
SPL {X  -165.650, Y  +461.106, Z    +0.000, E1   +30.916, E3 +446600.698}
SPL {X  -165.650, Y  +458.435, Z    +0.000, E1   +30.759, E3 +446610.906}
SPL {X  -165.650, Y  +454.220, Z    +0.000, E1   +30.954, E3 +446624.139}
SPL {X  -165.650, Y  +450.433, Z    +0.000, E1   +30.789, E3 +446638.104}
SPL {X  -165.650, Y  +447.097, Z    +0.000, E1   +30.843, E3 +446649.153}
SPL {X  -165.650, Y  +443.673, Z    +0.000, E1   +30.907, E3 +446660.460}
SPL {X  -165.650, Y  +440.976, Z    +0.000, E1   +30.719, E3 +446670.917}
SPL {X  -165.650, Y  +436.324, Z    +0.000, E1   +30.994, E3 +446685.203}
SPL {X  -165.650, Y  +432.765, Z    +0.000, E1   +30.831, E3 +446698.203}
SPL {X  -165.650, Y  +429.309, Z    +0.000, E1   +30.920, E3 +446709.544}
SPL {X  -165.650, Y  +424.918, Z    +0.000, E1   +30.862, E3 +446725.001}
SPL {X  -165.650, Y  +421.437, Z    +0.000, E1   +30.833, E3 +446736.970}
SPL {X  -165.650, Y  +417.366, Z    +0.000, E1   +30.879, E3 +446750.810}
SPL {X  -165.650, Y  +413.181, Z    +0.000, E1   +30.815, E3 +446765.408}
SPL {X  -165.650, Y  +408.547, Z    +0.000, E1   +30.964, E3 +446780.411}
SPL {X  -165.650, Y  +403.421, Z    +0.000, E1   +30.863, E3 +446798.628}
SPL {X  -165.650, Y  +398.147, Z    +0.000, E1   +30.902, E3 +446816.389}
SPL {X  -165.650, Y  +394.694, Z    +0.000, E1   +30.805, E3 +446828.697}
SPL {X  -165.650, Y  +390.331, Z    +0.000, E1   +30.892, E3 +446843.274}
SPL {X  -165.650, Y  +384.849, Z    +0.000, E1   +30.885, E3 +446862.077}
SPL {X  -165.650, Y  +380.752, Z    +0.000, E1   +30.927, E3 +446875.578}
SPL {X  -165.648, Y  +377.739, Z    +0.000, E1   +30.835, E3 +446886.588}
SPL {X  -165.594, Y  +374.183, Z    +0.000, E1   +30.878, E3 +446898.425}
SPL {X  -165.492, Y  +371.263, Z    +0.000, E1   +30.913, E3 +446908.120}
SPL {X  -165.379, Y  +369.027, Z    +0.000, E1   +30.727, E3 +446917.058}
SPL {X  -165.167, Y  +365.866, Z    +0.000, E1   +30.741, E3 +446927.832}
SPL {X  -164.892, Y  +362.671, Z    +0.000, E1   +30.830, E3 +446938.157}
SPL {X  -164.570, Y  +359.612, Z    +0.000, E1   +30.773, E3 +446948.969}
SPL {X  -164.104, Y  +355.923, Z    +0.000, E1   +30.626, E3 +446962.686}
SPL {X  -163.573, Y  +352.353, Z    +0.000, E1   +30.451, E3 +446975.950}
SPL {X  -162.476, Y  +346.230, Z    +0.000, E1   +31.677, E3 +446988.531}
SPL {X  -152.976, Y  +314.952, Z    +0.000, E1   +38.607, E3 +447037.496}
SPL {X  -137.967, Y  +286.821, Z    +0.000, E1   +43.969, E3 +447080.717}
ENDSPLINE

SPLINE
SPL {X  -153.316, Y  +315.777, Z    +0.000, E1   +33.140, E3 +447123.345}
SPL {X  -164.446, Y  +358.564, Z    +0.000, E1   +15.149, E3 +447088.556}
SPL {X  -165.379, Y  +369.025, Z    +0.000, E1    +9.158, E3 +447094.281}
SPL {X  -165.612, Y  +374.969, Z    +0.000, E1    +5.630, E3 +447096.956}
SPL {X  -165.650, Y  +383.362, Z    +0.000, E1    +0.177, E3 +447081.574}
SPL {X  -165.650, Y  +383.923, Z    +0.000, E1    -0.215, E3 +447094.732}
SPL {X  -165.650, Y  +388.083, Z    +0.000, E1    -3.355, E3 +447093.595}
SPL {X  -165.650, Y  +393.983, Z    +0.000, E1    -8.501, E3 +447089.994}
SPL {X  -165.650, Y  +402.241, Z    +0.000, E1   -16.711, E3 +447084.505}
SPL {X  -165.650, Y  +414.811, Z    +0.000, E1   -28.314, E3 +447084.036}
SPL {X  -165.650, Y  +423.479, Z    +0.000, E1   -29.012, E3 +447107.965}
SPL {X  -165.650, Y  +435.050, Z    +0.000, E1   -34.610, E3 +447116.299}
SPL {X  -165.650, Y  +446.725, Z    +0.000, E1   -39.593, E3 +447122.560}
SPL {X  -165.650, Y  +462.890, Z    +0.000, E1   -40.484, E3 +447153.736}
ENDSPLINE

SPLINE
SPL {X  -165.650, Y  +446.920, Z    +0.000, E1   -31.238, E3 +447166.062}
ENDSPLINE

SPLINE
SPL {X  -165.650, Y  +447.935, Z    +0.000, E1   -30.213, E3 +447176.350}
SPL {X  -165.650, Y  +451.020, Z    +0.000, E1   -30.224, E3 +447187.170}
SPL {X  -165.650, Y  +454.519, Z    +0.000, E1   -30.374, E3 +447198.353}
SPL {X  -165.650, Y  +456.542, Z    +0.000, E1   -29.986, E3 +447208.098}
SPL {X  -165.650, Y  +460.618, Z    +0.000, E1   -30.298, E3 +447220.418}
SPL {X  -165.650, Y  +463.853, Z    +0.000, E1   -30.103, E3 +447233.019}
SPL {X  -165.650, Y  +467.246, Z    +0.000, E1   -30.279, E3 +447243.749}
SPL {X  -165.650, Y  +469.780, Z    +0.000, E1   -30.237, E3 +447252.874}
SPL {X  -165.650, Y  +472.566, Z    +0.000, E1   -30.124, E3 +447263.532}
SPL {X  -165.650, Y  +476.540, Z    +0.000, E1   -30.193, E3 +447277.076}
SPL {X  -165.650, Y  +480.320, Z    +0.000, E1   -30.163, E3 +447290.554}
SPL {X  -165.650, Y  +484.477, Z    +0.000, E1   -30.274, E3 +447304.443}
SPL {X  -165.650, Y  +489.057, Z    +0.000, E1   -30.341, E3 +447320.083}
SPL {X  -165.650, Y  +491.647, Z    +0.000, E1   -29.894, E3 +447332.016}
SPL {X  -165.650, Y  +495.051, Z    +0.000, E1   -30.213, E3 +447341.945}
SPL {X  -165.650, Y  +499.546, Z    +0.000, E1   -30.283, E3 +447357.388}
SPL {X  -165.650, Y  +503.544, Z    +0.000, E1   -30.247, E3 +447371.456}
SPL {X  -165.650, Y  +506.344, Z    +0.000, E1   -30.129, E3 +447382.125}
SPL {X  -165.650, Y  +510.660, Z    +0.000, E1   -30.223, E3 +447396.828}
SPL {X  -165.650, Y  +515.918, Z    +0.000, E1   -30.316, E3 +447414.637}
SPL {X  -165.650, Y  +520.621, Z    +0.000, E1   -30.198, E3 +447431.922}
SPL {X  -165.650, Y  +525.344, Z    +0.000, E1   -30.269, E3 +447447.979}
SPL {X  -165.650, Y  +528.152, Z    +0.000, E1   -29.991, E3 +447459.619}
SPL {X  -165.650, Y  +531.783, Z    +0.000, E1   -30.416, E3 +447469.512}
SPL {X  -165.650, Y  +534.115, Z    +0.000, E1   -30.089, E3 +447479.894}
SPL {X  -165.650, Y  +537.522, Z    +0.000, E1   -30.251, E3 +447490.809}
SPL {X  -165.650, Y  +540.621, Z    +0.000, E1   -30.014, E3 +447503.370}
SPL {X  -165.650, Y  +544.944, Z    +0.000, E1   -30.447, E3 +447515.569}
SPL {X  -165.650, Y  +547.199, Z    +0.000, E1   -30.132, E3 +447525.543}
SPL {X  -165.650, Y  +550.512, Z    +0.000, E1   -30.197, E3 +447536.869}
SPL {X  -165.650, Y  +553.852, Z    +0.000, E1   -30.156, E3 +447548.809}
SPL {X  -165.650, Y  +557.277, Z    +0.000, E1   -30.150, E3 +447560.984}
SPL {X  -165.650, Y  +561.168, Z    +0.000, E1   -30.194, E3 +447574.365}
SPL {X  -165.650, Y  +564.449, Z    +0.000, E1   -30.167, E3 +447586.049}
SPL {X  -165.650, Y  +566.935, Z    +0.000, E1   -30.135, E3 +447594.954}
SPL {X  -165.650, Y  +570.048, Z    +0.000, E1   -30.238, E3 +447605.279}
SPL {X  -165.650, Y  +573.110, Z    +0.000, E1   -30.057, E3 +447617.264}
SPL {X  -165.650, Y  +577.587, Z    +0.000, E1   -30.270, E3 +447631.703}
SPL {X  -165.650, Y  +581.190, Z    +0.000, E1   -30.107, E3 +447645.342}
SPL {X  -165.650, Y  +585.096, Z    +0.000, E1   -30.203, E3 +447658.529}
ENDSPLINE

SPLINE
SPL {X  -165.650, Y  +584.346, Z    +0.000, E1   -28.397, E3 +447667.876}
SPL {X  -165.650, Y  +484.445, Z    +0.000, E1   +32.277, E3 +447676.617}
SPL {X  -165.650, Y  +481.524, Z    +0.000, E1   +31.089, E3 +447694.068}
SPL {X  -165.650, Y  +478.014, Z    +0.000, E1   +30.826, E3 +447707.675}
SPL {X  -165.650, Y  +474.473, Z    +0.000, E1   +30.943, E3 +447719.000}
SPL {X  -165.650, Y  +471.826, Z    +0.000, E1   +30.770, E3 +447729.183}
SPL {X  -165.650, Y  +467.753, Z    +0.000, E1   +30.878, E3 +447742.557}
SPL {X  -165.650, Y  +463.837, Z    +0.000, E1   +30.924, E3 +447755.490}
SPL {X  -165.650, Y  +461.106, Z    +0.000, E1   +30.916, E3 +447764.877}
SPL {X  -165.650, Y  +458.435, Z    +0.000, E1   +30.759, E3 +447775.085}
SPL {X  -165.650, Y  +454.220, Z    +0.000, E1   +30.954, E3 +447788.318}
SPL {X  -165.650, Y  +450.433, Z    +0.000, E1   +30.789, E3 +447802.283}
SPL {X  -165.650, Y  +447.097, Z    +0.000, E1   +30.843, E3 +447813.332}
SPL {X  -165.650, Y  +443.673, Z    +0.000, E1   +30.907, E3 +447824.639}
SPL {X  -165.650, Y  +440.976, Z    +0.000, E1   +30.719, E3 +447835.096}
SPL {X  -165.650, Y  +436.324, Z    +0.000, E1   +30.994, E3 +447849.383}
SPL {X  -165.650, Y  +432.765, Z    +0.000, E1   +30.831, E3 +447862.383}
SPL {X  -165.650, Y  +429.309, Z    +0.000, E1   +30.920, E3 +447873.723}
SPL {X  -165.650, Y  +424.918, Z    +0.000, E1   +30.862, E3 +447889.180}
SPL {X  -165.650, Y  +421.437, Z    +0.000, E1   +30.833, E3 +447901.149}
SPL {X  -165.650, Y  +417.366, Z    +0.000, E1   +30.879, E3 +447914.989}
SPL {X  -165.650, Y  +413.181, Z    +0.000, E1   +30.815, E3 +447929.587}
SPL {X  -165.650, Y  +408.547, Z    +0.000, E1   +30.964, E3 +447944.590}
SPL {X  -165.650, Y  +403.421, Z    +0.000, E1   +30.863, E3 +447962.807}
SPL {X  -165.650, Y  +398.147, Z    +0.000, E1   +30.902, E3 +447980.568}
SPL {X  -165.650, Y  +394.694, Z    +0.000, E1   +30.805, E3 +447992.876}
SPL {X  -165.650, Y  +390.331, Z    +0.000, E1   +30.892, E3 +448007.453}
SPL {X  -165.650, Y  +384.849, Z    +0.000, E1   +30.885, E3 +448026.256}
SPL {X  -165.650, Y  +380.752, Z    +0.000, E1   +30.927, E3 +448039.758}
SPL {X  -165.648, Y  +377.739, Z    +0.000, E1   +30.835, E3 +448050.767}
SPL {X  -165.594, Y  +374.183, Z    +0.000, E1   +30.878, E3 +448062.604}
SPL {X  -165.492, Y  +371.263, Z    +0.000, E1   +30.913, E3 +448072.299}
SPL {X  -165.379, Y  +369.027, Z    +0.000, E1   +30.727, E3 +448081.237}
SPL {X  -165.167, Y  +365.866, Z    +0.000, E1   +30.741, E3 +448092.012}
SPL {X  -164.892, Y  +362.671, Z    +0.000, E1   +30.830, E3 +448102.336}
SPL {X  -164.570, Y  +359.612, Z    +0.000, E1   +30.773, E3 +448113.148}
SPL {X  -164.104, Y  +355.923, Z    +0.000, E1   +30.626, E3 +448126.865}
SPL {X  -163.573, Y  +352.353, Z    +0.000, E1   +30.451, E3 +448140.130}
SPL {X  -162.476, Y  +346.230, Z    +0.000, E1   +31.677, E3 +448152.710}
SPL {X  -152.976, Y  +314.952, Z    +0.000, E1   +38.607, E3 +448201.675}
SPL {X  -137.967, Y  +286.821, Z    +0.000, E1   +43.969, E3 +448244.897}
ENDSPLINE

SPLINE
SPL {X  -153.316, Y  +315.777, Z    +0.000, E1   +33.140, E3 +448287.524}
SPL {X  -164.446, Y  +358.564, Z    +0.000, E1   +15.149, E3 +448252.735}
SPL {X  -165.510, Y  +371.680, Z    +0.000, E1    +7.684, E3 +448256.790}
SPL {X  -165.628, Y  +375.818, Z    +0.000, E1    +5.016, E3 +448264.720}
SPL {X  -165.650, Y  +383.362, Z    +0.000, E1    +0.177, E3 +448245.754}
SPL {X  -165.650, Y  +383.923, Z    +0.000, E1    -0.215, E3 +448258.911}
SPL {X  -165.650, Y  +388.083, Z    +0.000, E1    -3.355, E3 +448257.774}
SPL {X  -165.650, Y  +393.983, Z    +0.000, E1    -8.501, E3 +448254.173}
SPL {X  -165.650, Y  +402.241, Z    +0.000, E1   -16.711, E3 +448248.684}
SPL {X  -165.650, Y  +414.811, Z    +0.000, E1   -28.314, E3 +448248.215}
SPL {X  -165.650, Y  +423.479, Z    +0.000, E1   -29.012, E3 +448272.144}
SPL {X  -165.650, Y  +441.276, Z    +0.000, E1   -37.343, E3 +448283.833}
SPL {X  -165.650, Y  +462.890, Z    +0.000, E1   -40.484, E3 +448317.915}
ENDSPLINE

SPLINE
SPL {X  -165.650, Y  +446.920, Z    +0.000, E1   -31.238, E3 +448330.241}
ENDSPLINE

SPLINE
SPL {X  -165.650, Y  +447.935, Z    +0.000, E1   -30.213, E3 +448340.529}
SPL {X  -165.650, Y  +451.020, Z    +0.000, E1   -30.224, E3 +448351.350}
SPL {X  -165.650, Y  +454.519, Z    +0.000, E1   -30.374, E3 +448362.532}
SPL {X  -165.650, Y  +457.429, Z    +0.000, E1   -30.029, E3 +448375.234}
SPL {X  -165.650, Y  +461.678, Z    +0.000, E1   -30.426, E3 +448387.358}
SPL {X  -165.650, Y  +463.853, Z    +0.000, E1   -30.103, E3 +448397.198}
SPL {X  -165.650, Y  +468.397, Z    +0.000, E1   -30.302, E3 +448412.002}
SPL {X  -165.650, Y  +472.566, Z    +0.000, E1   -30.124, E3 +448427.711}
SPL {X  -165.650, Y  +476.540, Z    +0.000, E1   -30.193, E3 +448441.255}
SPL {X  -165.650, Y  +481.042, Z    +0.000, E1   -30.192, E3 +448457.200}
SPL {X  -165.650, Y  +485.236, Z    +0.000, E1   -30.294, E3 +448471.056}
SPL {X  -165.650, Y  +489.057, Z    +0.000, E1   -30.341, E3 +448484.262}
SPL {X  -165.650, Y  +491.647, Z    +0.000, E1   -29.894, E3 +448496.195}
SPL {X  -165.650, Y  +495.051, Z    +0.000, E1   -30.213, E3 +448506.124}
SPL {X  -165.650, Y  +498.418, Z    +0.000, E1   -30.282, E3 +448517.417}
SPL {X  -165.650, Y  +502.421, Z    +0.000, E1   -30.263, E3 +448531.774}
SPL {X  -165.650, Y  +506.344, Z    +0.000, E1   -30.129, E3 +448546.304}
SPL {X  -165.650, Y  +509.866, Z    +0.000, E1   -30.236, E3 +448557.973}
SPL {X  -165.650, Y  +513.685, Z    +0.000, E1   -30.234, E3 +448571.470}
SPL {X  -165.650, Y  +517.919, Z    +0.000, E1   -30.227, E3 +448586.377}
SPL {X  -165.650, Y  +521.521, Z    +0.000, E1   -30.210, E3 +448599.051}
SPL {X  -165.650, Y  +525.344, Z    +0.000, E1   -30.269, E3 +448612.158}
SPL {X  -165.650, Y  +528.152, Z    +0.000, E1   -29.991, E3 +448623.799}
SPL {X  -165.650, Y  +531.783, Z    +0.000, E1   -30.416, E3 +448633.691}
SPL {X  -165.650, Y  +534.115, Z    +0.000, E1   -30.089, E3 +448644.073}
SPL {X  -165.650, Y  +537.522, Z    +0.000, E1   -30.251, E3 +448654.988}
SPL {X  -165.650, Y  +540.621, Z    +0.000, E1   -30.014, E3 +448667.549}
SPL {X  -165.650, Y  +544.944, Z    +0.000, E1   -30.447, E3 +448679.748}
SPL {X  -165.650, Y  +548.549, Z    +0.000, E1   -30.216, E3 +448694.072}
SPL {X  -165.650, Y  +553.092, Z    +0.000, E1   -30.157, E3 +448710.414}
SPL {X  -165.650, Y  +556.274, Z    +0.000, E1   -30.127, E3 +448721.669}
SPL {X  -165.650, Y  +560.243, Z    +0.000, E1   -30.214, E3 +448735.335}
SPL {X  -165.650, Y  +565.528, Z    +0.000, E1   -30.192, E3 +448754.027}
SPL {X  -165.650, Y  +570.048, Z    +0.000, E1   -30.238, E3 +448769.458}
SPL {X  -165.650, Y  +573.110, Z    +0.000, E1   -30.057, E3 +448781.443}
SPL {X  -165.650, Y  +577.587, Z    +0.000, E1   -30.270, E3 +448795.882}
SPL {X  -165.650, Y  +581.190, Z    +0.000, E1   -30.107, E3 +448809.522}
SPL {X  -165.650, Y  +585.053, Z    +0.000, E1   -30.090, E3 +448823.392}
ENDSPLINE

SPLINE
SPL {X  -165.650, Y  +484.445, Z    +0.000, E1   +32.277, E3 +448840.796}
SPL {X  -165.650, Y  +481.524, Z    +0.000, E1   +31.089, E3 +448858.247}
SPL {X  -165.650, Y  +478.014, Z    +0.000, E1   +30.826, E3 +448871.854}
SPL {X  -165.650, Y  +474.473, Z    +0.000, E1   +30.943, E3 +448883.179}
SPL {X  -165.650, Y  +471.826, Z    +0.000, E1   +30.770, E3 +448893.362}
SPL {X  -165.650, Y  +467.753, Z    +0.000, E1   +30.878, E3 +448906.736}
SPL {X  -165.650, Y  +463.837, Z    +0.000, E1   +30.924, E3 +448919.670}
SPL {X  -165.650, Y  +461.106, Z    +0.000, E1   +30.916, E3 +448929.056}
SPL {X  -165.650, Y  +457.156, Z    +0.000, E1   +30.860, E3 +448943.133}
SPL {X  -165.650, Y  +453.156, Z    +0.000, E1   +30.934, E3 +448956.107}
SPL {X  -165.650, Y  +450.433, Z    +0.000, E1   +30.789, E3 +448966.462}
SPL {X  -165.650, Y  +447.097, Z    +0.000, E1   +30.843, E3 +448977.511}
SPL {X  -165.650, Y  +443.673, Z    +0.000, E1   +30.907, E3 +448988.818}
SPL {X  -165.650, Y  +439.486, Z    +0.000, E1   +30.857, E3 +449003.628}
SPL {X  -165.650, Y  +434.043, Z    +0.000, E1   +30.950, E3 +449021.644}
SPL {X  -165.650, Y  +430.419, Z    +0.000, E1   +30.895, E3 +449034.147}
SPL {X  -165.650, Y  +427.340, Z    +0.000, E1   +30.870, E3 +449044.974}
SPL {X  -165.650, Y  +422.641, Z    +0.000, E1   +30.884, E3 +449061.063}
SPL {X  -165.650, Y  +417.366, Z    +0.000, E1   +30.879, E3 +449079.168}
SPL {X  -165.650, Y  +412.139, Z    +0.000, E1   +30.870, E3 +449097.118}
SPL {X  -165.650, Y  +406.834, Z    +0.000, E1   +30.919, E3 +449114.947}
SPL {X  -165.650, Y  +402.516, Z    +0.000, E1   +30.874, E3 +449129.869}
SPL {X  -165.650, Y  +398.147, Z    +0.000, E1   +30.902, E3 +449144.747}
SPL {X  -165.650, Y  +394.694, Z    +0.000, E1   +30.805, E3 +449157.056}
SPL {X  -165.650, Y  +391.522, Z    +0.000, E1   +30.837, E3 +449167.736}
SPL {X  -165.650, Y  +387.533, Z    +0.000, E1   +30.858, E3 +449181.363}
SPL {X  -165.650, Y  +383.627, Z    +0.000, E1   +30.885, E3 +449194.423}
SPL {X  -165.650, Y  +380.752, Z    +0.000, E1   +30.927, E3 +449203.937}
SPL {X  -165.648, Y  +377.739, Z    +0.000, E1   +30.835, E3 +449214.946}
SPL {X  -165.594, Y  +374.183, Z    +0.000, E1   +30.878, E3 +449226.783}
SPL {X  -165.492, Y  +371.263, Z    +0.000, E1   +30.913, E3 +449236.478}
SPL {X  -165.379, Y  +369.027, Z    +0.000, E1   +30.727, E3 +449245.417}
SPL {X  -165.167, Y  +365.866, Z    +0.000, E1   +30.741, E3 +449256.191}
SPL {X  -164.892, Y  +362.671, Z    +0.000, E1   +30.830, E3 +449266.515}
SPL {X  -164.570, Y  +359.612, Z    +0.000, E1   +30.773, E3 +449277.327}
SPL {X  -164.104, Y  +355.923, Z    +0.000, E1   +30.626, E3 +449291.044}
SPL {X  -163.573, Y  +352.353, Z    +0.000, E1   +30.451, E3 +449304.309}
SPL {X  -162.976, Y  +348.856, Z    +0.000, E1   +30.757, E3 +449314.232}
SPL {X  -161.497, Y  +341.640, Z    +0.000, E1   +33.276, E3 +449321.510}
SPL {X  -152.976, Y  +314.952, Z    +0.000, E1   +38.607, E3 +449365.855}
SPL {X  -137.967, Y  +286.821, Z    +0.000, E1   +43.969, E3 +449409.076}
ENDSPLINE

SPLINE
SPL {X  -149.143, Y  +306.414, Z    +0.000, E1   +36.361, E3 +449460.208}
SPL {X  -163.091, Y  +349.496, Z    +0.000, E1   +19.699, E3 +449416.991}
SPL {X  -164.704, Y  +360.824, Z    +0.000, E1   +13.856, E3 +449418.332}
SPL {X  -165.510, Y  +371.680, Z    +0.000, E1    +7.684, E3 +449420.970}
SPL {X  -165.628, Y  +375.818, Z    +0.000, E1    +5.016, E3 +449428.899}
SPL {X  -165.650, Y  +383.362, Z    +0.000, E1    +0.177, E3 +449409.933}
SPL {X  -165.650, Y  +383.923, Z    +0.000, E1    -0.215, E3 +449423.090}
SPL {X  -165.650, Y  +388.083, Z    +0.000, E1    -3.355, E3 +449421.954}
SPL {X  -165.650, Y  +393.983, Z    +0.000, E1    -8.501, E3 +449418.352}
SPL {X  -165.650, Y  +402.241, Z    +0.000, E1   -16.711, E3 +449412.864}
SPL {X  -165.650, Y  +416.345, Z    +0.000, E1   -29.511, E3 +449412.656}
SPL {X  -165.650, Y  +422.331, Z    +0.000, E1   -27.760, E3 +449438.155}
SPL {X  -165.650, Y  +441.276, Z    +0.000, E1   -37.343, E3 +449448.012}
SPL {X  -165.650, Y  +462.890, Z    +0.000, E1   -40.484, E3 +449482.095}
ENDSPLINE

SPLINE
SPL {X  -165.650, Y  +446.920, Z    +0.000, E1   -31.238, E3 +449494.420}
ENDSPLINE

SPLINE
SPL {X  -165.650, Y  +447.935, Z    +0.000, E1   -30.213, E3 +449504.708}
SPL {X  -165.650, Y  +451.020, Z    +0.000, E1   -30.224, E3 +449515.529}
SPL {X  -165.650, Y  +454.519, Z    +0.000, E1   -30.374, E3 +449526.711}
SPL {X  -165.650, Y  +456.542, Z    +0.000, E1   -29.986, E3 +449536.456}
SPL {X  -165.650, Y  +460.618, Z    +0.000, E1   -30.298, E3 +449548.776}
SPL {X  -165.650, Y  +463.853, Z    +0.000, E1   -30.103, E3 +449561.377}
SPL {X  -165.650, Y  +467.246, Z    +0.000, E1   -30.279, E3 +449572.107}
SPL {X  -165.650, Y  +469.780, Z    +0.000, E1   -30.237, E3 +449581.233}
SPL {X  -165.650, Y  +472.566, Z    +0.000, E1   -30.124, E3 +449591.890}
SPL {X  -165.650, Y  +476.540, Z    +0.000, E1   -30.193, E3 +449605.434}
SPL {X  -165.650, Y  +481.042, Z    +0.000, E1   -30.192, E3 +449621.380}
SPL {X  -165.650, Y  +485.236, Z    +0.000, E1   -30.294, E3 +449635.235}
SPL {X  -165.650, Y  +488.041, Z    +0.000, E1   -30.253, E3 +449645.356}
SPL {X  -165.650, Y  +491.281, Z    +0.000, E1   -30.148, E3 +449657.495}
SPL {X  -165.650, Y  +495.051, Z    +0.000, E1   -30.213, E3 +449670.303}
SPL {X  -165.650, Y  +498.418, Z    +0.000, E1   -30.282, E3 +449681.596}
SPL {X  -165.650, Y  +502.421, Z    +0.000, E1   -30.263, E3 +449695.953}
SPL {X  -165.650, Y  +506.344, Z    +0.000, E1   -30.129, E3 +449710.483}
SPL {X  -165.650, Y  +510.660, Z    +0.000, E1   -30.223, E3 +449725.187}
SPL {X  -165.650, Y  +515.918, Z    +0.000, E1   -30.316, E3 +449742.995}
SPL {X  -165.650, Y  +520.621, Z    +0.000, E1   -30.198, E3 +449760.280}
SPL {X  -165.650, Y  +525.344, Z    +0.000, E1   -30.269, E3 +449776.337}
SPL {X  -165.650, Y  +528.152, Z    +0.000, E1   -29.991, E3 +449787.978}
SPL {X  -165.650, Y  +531.783, Z    +0.000, E1   -30.416, E3 +449797.870}
SPL {X  -165.650, Y  +534.115, Z    +0.000, E1   -30.089, E3 +449808.253}
SPL {X  -165.650, Y  +538.363, Z    +0.000, E1   -30.232, E3 +449822.422}
SPL {X  -165.650, Y  +543.650, Z    +0.000, E1   -30.281, E3 +449840.642}
SPL {X  -165.650, Y  +547.199, Z    +0.000, E1   -30.132, E3 +449853.901}
SPL {X  -165.650, Y  +550.512, Z    +0.000, E1   -30.197, E3 +449865.227}
SPL {X  -165.650, Y  +554.908, Z    +0.000, E1   -30.180, E3 +449880.888}
SPL {X  -165.650, Y  +560.243, Z    +0.000, E1   -30.214, E3 +449899.514}
SPL {X  -165.650, Y  +565.528, Z    +0.000, E1   -30.192, E3 +449918.206}
SPL {X  -165.650, Y  +570.048, Z    +0.000, E1   -30.238, E3 +449933.637}
SPL {X  -165.650, Y  +573.110, Z    +0.000, E1   -30.057, E3 +449945.622}
SPL {X  -165.650, Y  +577.587, Z    +0.000, E1   -30.270, E3 +449960.061}
SPL {X  -165.650, Y  +581.190, Z    +0.000, E1   -30.107, E3 +449973.701}
SPL {X  -165.650, Y  +585.053, Z    +0.000, E1   -30.090, E3 +449987.571}
ENDSPLINE

SPLINE
SPL {X  -165.650, Y  +484.968, Z    +0.000, E1   +32.508, E3 +450001.537}
SPL {X  -165.650, Y  +482.280, Z    +0.000, E1   +31.680, E3 +450015.863}
SPL {X  -165.650, Y  +479.331, Z    +0.000, E1   +30.680, E3 +450032.611}
SPL {X  -165.650, Y  +474.473, Z    +0.000, E1   +30.943, E3 +450047.358}
SPL {X  -165.650, Y  +471.826, Z    +0.000, E1   +30.770, E3 +450057.541}
SPL {X  -165.650, Y  +467.753, Z    +0.000, E1   +30.878, E3 +450070.915}
SPL {X  -165.650, Y  +463.837, Z    +0.000, E1   +30.924, E3 +450083.849}
SPL {X  -165.650, Y  +461.106, Z    +0.000, E1   +30.916, E3 +450093.236}
SPL {X  -165.650, Y  +457.156, Z    +0.000, E1   +30.860, E3 +450107.312}
SPL {X  -165.650, Y  +453.156, Z    +0.000, E1   +30.934, E3 +450120.286}
SPL {X  -165.650, Y  +450.433, Z    +0.000, E1   +30.789, E3 +450130.641}
SPL {X  -165.650, Y  +447.097, Z    +0.000, E1   +30.843, E3 +450141.690}
SPL {X  -165.650, Y  +443.673, Z    +0.000, E1   +30.907, E3 +450152.998}
SPL {X  -165.650, Y  +439.486, Z    +0.000, E1   +30.857, E3 +450167.807}
SPL {X  -165.650, Y  +435.146, Z    +0.000, E1   +30.969, E3 +450181.726}
SPL {X  -165.650, Y  +431.607, Z    +0.000, E1   +30.889, E3 +450194.441}
SPL {X  -165.650, Y  +427.340, Z    +0.000, E1   +30.870, E3 +450209.153}
SPL {X  -165.650, Y  +423.901, Z    +0.000, E1   +30.858, E3 +450220.909}
SPL {X  -165.650, Y  +421.437, Z    +0.000, E1   +30.833, E3 +450229.507}
SPL {X  -165.650, Y  +418.489, Z    +0.000, E1   +30.835, E3 +450239.624}
SPL {X  -165.650, Y  +414.127, Z    +0.000, E1   +30.869, E3 +450254.532}
SPL {X  -165.650, Y  +408.547, Z    +0.000, E1   +30.964, E3 +450272.948}
SPL {X  -165.650, Y  +405.433, Z    +0.000, E1   +30.730, E3 +450284.925}
SPL {X  -165.650, Y  +401.473, Z    +0.000, E1   +30.933, E3 +450297.374}
SPL {X  -165.650, Y  +396.018, Z    +0.000, E1   +30.861, E3 +450316.558}
SPL {X  -165.650, Y  +391.522, Z    +0.000, E1   +30.837, E3 +450331.915}
SPL {X  -165.650, Y  +387.533, Z    +0.000, E1   +30.858, E3 +450345.542}
SPL {X  -165.650, Y  +383.627, Z    +0.000, E1   +30.885, E3 +450358.602}
SPL {X  -165.650, Y  +380.752, Z    +0.000, E1   +30.927, E3 +450368.116}
SPL {X  -165.648, Y  +377.739, Z    +0.000, E1   +30.835, E3 +450379.125}
SPL {X  -165.594, Y  +374.183, Z    +0.000, E1   +30.878, E3 +450390.962}
SPL {X  -165.429, Y  +369.945, Z    +0.000, E1   +30.850, E3 +450405.837}
SPL {X  -165.167, Y  +365.866, Z    +0.000, E1   +30.741, E3 +450420.370}
SPL {X  -164.892, Y  +362.671, Z    +0.000, E1   +30.830, E3 +450430.694}
SPL {X  -164.570, Y  +359.612, Z    +0.000, E1   +30.773, E3 +450441.506}
SPL {X  -164.104, Y  +355.923, Z    +0.000, E1   +30.626, E3 +450455.223}
SPL {X  -163.573, Y  +352.353, Z    +0.000, E1   +30.451, E3 +450468.488}
SPL {X  -162.476, Y  +346.230, Z    +0.000, E1   +31.677, E3 +450481.069}
SPL {X  -152.976, Y  +314.952, Z    +0.000, E1   +38.607, E3 +450530.034}
SPL {X  -137.967, Y  +286.821, Z    +0.000, E1   +43.969, E3 +450573.255}
ENDSPLINE

SPLINE
SPL {X  -153.316, Y  +315.777, Z    +0.000, E1   +33.140, E3 +450615.882}
SPL {X  -164.446, Y  +358.564, Z    +0.000, E1   +15.149, E3 +450581.093}
SPL {X  -165.379, Y  +369.025, Z    +0.000, E1    +9.158, E3 +450586.818}
SPL {X  -165.612, Y  +374.969, Z    +0.000, E1    +5.630, E3 +450589.493}
SPL {X  -165.650, Y  +383.362, Z    +0.000, E1    +0.177, E3 +450574.112}
SPL {X  -165.650, Y  +383.923, Z    +0.000, E1    -0.215, E3 +450587.269}
SPL {X  -165.650, Y  +388.083, Z    +0.000, E1    -3.355, E3 +450586.133}
SPL {X  -165.650, Y  +393.983, Z    +0.000, E1    -8.501, E3 +450582.531}
SPL {X  -165.650, Y  +402.241, Z    +0.000, E1   -16.711, E3 +450577.043}
SPL {X  -165.650, Y  +416.345, Z    +0.000, E1   -29.511, E3 +450576.835}
SPL {X  -165.650, Y  +422.331, Z    +0.000, E1   -27.760, E3 +450602.334}
SPL {X  -165.650, Y  +441.276, Z    +0.000, E1   -37.343, E3 +450612.191}
SPL {X  -165.650, Y  +462.890, Z    +0.000, E1   -40.484, E3 +450646.274}
ENDSPLINE

SPLINE
SPL {X  -165.650, Y  +446.920, Z    +0.000, E1   -31.238, E3 +450658.600}
ENDSPLINE

SPLINE
SPL {X  -165.650, Y  +447.935, Z    +0.000, E1   -30.213, E3 +450668.887}
SPL {X  -165.650, Y  +451.020, Z    +0.000, E1   -30.224, E3 +450679.708}
SPL {X  -165.650, Y  +454.519, Z    +0.000, E1   -30.374, E3 +450690.890}
SPL {X  -165.650, Y  +456.542, Z    +0.000, E1   -29.986, E3 +450700.635}
SPL {X  -165.650, Y  +460.618, Z    +0.000, E1   -30.298, E3 +450712.955}
SPL {X  -165.650, Y  +463.853, Z    +0.000, E1   -30.103, E3 +450725.556}
SPL {X  -165.650, Y  +467.246, Z    +0.000, E1   -30.279, E3 +450736.286}
SPL {X  -165.650, Y  +469.780, Z    +0.000, E1   -30.237, E3 +450745.412}
SPL {X  -165.650, Y  +472.566, Z    +0.000, E1   -30.124, E3 +450756.069}
SPL {X  -165.650, Y  +476.540, Z    +0.000, E1   -30.193, E3 +450769.613}
SPL {X  -165.650, Y  +480.320, Z    +0.000, E1   -30.163, E3 +450783.091}
SPL {X  -165.650, Y  +484.477, Z    +0.000, E1   -30.274, E3 +450796.980}
SPL {X  -165.650, Y  +488.041, Z    +0.000, E1   -30.253, E3 +450809.536}
SPL {X  -165.650, Y  +491.281, Z    +0.000, E1   -30.148, E3 +450821.674}
SPL {X  -165.650, Y  +495.051, Z    +0.000, E1   -30.213, E3 +450834.482}
SPL {X  -165.650, Y  +498.418, Z    +0.000, E1   -30.282, E3 +450845.775}
SPL {X  -165.650, Y  +500.833, Z    +0.000, E1   -30.191, E3 +450854.824}
SPL {X  -165.650, Y  +504.246, Z    +0.000, E1   -30.231, E3 +450866.690}
SPL {X  -165.650, Y  +507.017, Z    +0.000, E1   -30.108, E3 +450877.099}
SPL {X  -165.650, Y  +510.660, Z    +0.000, E1   -30.223, E3 +450889.366}
SPL {X  -165.650, Y  +514.670, Z    +0.000, E1   -30.278, E3 +450902.875}
SPL {X  -165.650, Y  +517.919, Z    +0.000, E1   -30.227, E3 +450914.735}
SPL {X  -165.650, Y  +521.521, Z    +0.000, E1   -30.210, E3 +450927.410}
SPL {X  -165.650, Y  +525.344, Z    +0.000, E1   -30.269, E3 +450940.516}
SPL {X  -165.650, Y  +528.152, Z    +0.000, E1   -29.991, E3 +450952.157}
SPL {X  -165.650, Y  +531.783, Z    +0.000, E1   -30.416, E3 +450962.050}
SPL {X  -165.650, Y  +534.115, Z    +0.000, E1   -30.089, E3 +450972.432}
SPL {X  -165.650, Y  +537.522, Z    +0.000, E1   -30.251, E3 +450983.346}
SPL {X  -165.650, Y  +540.621, Z    +0.000, E1   -30.014, E3 +450995.907}
SPL {X  -165.650, Y  +544.944, Z    +0.000, E1   -30.447, E3 +451008.107}
SPL {X  -165.650, Y  +547.199, Z    +0.000, E1   -30.132, E3 +451018.080}
SPL {X  -165.650, Y  +550.512, Z    +0.000, E1   -30.197, E3 +451029.406}
SPL {X  -165.650, Y  +553.852, Z    +0.000, E1   -30.156, E3 +451041.347}
SPL {X  -165.650, Y  +557.277, Z    +0.000, E1   -30.150, E3 +451053.521}
SPL {X  -165.650, Y  +561.168, Z    +0.000, E1   -30.194, E3 +451066.903}
SPL {X  -165.650, Y  +564.449, Z    +0.000, E1   -30.167, E3 +451078.586}
SPL {X  -165.650, Y  +566.935, Z    +0.000, E1   -30.135, E3 +451087.491}
SPL {X  -165.650, Y  +570.048, Z    +0.000, E1   -30.238, E3 +451097.816}
SPL {X  -165.650, Y  +573.110, Z    +0.000, E1   -30.057, E3 +451109.801}
SPL {X  -165.650, Y  +577.587, Z    +0.000, E1   -30.270, E3 +451124.240}
SPL {X  -165.650, Y  +581.190, Z    +0.000, E1   -30.107, E3 +451137.880}
SPL {X  -165.650, Y  +585.053, Z    +0.000, E1   -30.090, E3 +451151.750}
ENDSPLINE

